// SIMATIC STEP 7 (V5.x) project PLC_PKS
// CPU: CPU 315-2 PN/DP
// station: Hardware
// station: SIMATIC 300
// station: P_ADR_BUS
// program: S7 Program(1)

SYMBOL_TABLE
"CV1_pid"	DB 2	FB 2
"COM"	DB 88	DB 88
"COMM"	DB 100	DB 100
"CV1_ctrl"	DB 201	FB 2
"CV6_ctrl"	DB 206	FB 2
"CV7_ctrl"	DB 207	FB 2
"CV8_ctrl"	DB 208	FB 2
"CV9_ctrl"	DB 209	FB 2
"CV10_ctrl"	DB 210	FB 2
"CV11_ctrl"	DB 211	FB 2
"CV12_ctrl"	DB 212	FB 2
"CV13_ctrl"	DB 213	FB 2
"CV14_ctrl"	DB 214	FB 2
"CV15_ctrl"	DB 215	FB 2
"CV16_ctrl"	DB 216	FB 2
"CV17_ctrl"	DB 217	FB 2
"CV18_1_ctrl"	DB 218	FB 2
"CV18_2_ctrl"	DB 219	FB 2
"CV21_ctrl"	DB 221	FB 2
"CV22_ctrl"	DB 222	FB 2
"ctrl_CV23"	DB 223	FB 2
"ctrl_CV24"	DB 224	FB 2
"ctrl_CV25"	DB 225	FB 2
"pid_cv1"	DB 501	FB 58
"pid_cv2"	DB 502	FB 58
"pid_cv6"	DB 506	FB 58
"pid_cv7"	DB 507	FB 58
"pid_cv8"	DB 508	FB 58
"pid_cv9"	DB 509	FB 58
"pid_cv10"	DB 510	FB 58
"pid_cv11"	DB 511	FB 58
"pid_cv12"	DB 512	FB 58
"pid_cv13"	DB 513	FB 58
"pid_cv14"	DB 514	FB 58
"pid_cv15"	DB 515	FB 58
"pid_cv16"	DB 516	FB 58
"pid_cv17"	DB 517	FB 58
"pid_cv18_1"	DB 518	FB 58
"pid_cv18_2"	DB 519	FB 58
"pid_cv21"	DB 521	FB 58
"pid_cv22"	DB 522	FB 58
"pid_cv23"	DB 523	FB 58
"pid_cv24"	DB 524	FB 58
"pid_cv25"	DB 525	FB 58
"Pumps"	FB 1	FB 1
"klapan"	FB 2	FB 2
"Dat_CV_val"	FB 3	FB 3
"TCONT_CP"	FB 58	FB 58	// temperature PID controller with pulse generator and self-tuning
"Dat_Filt"	FC 1	FC 1
"SCALE"	FC 105	FC 105	// Scaling Values
"UNSCALE"	FC 106	FC 106	// Unscaling Values
"MM1_KM"	M 10.0	BOOL
"M1_Man"	M 1424.0	BOOL
"CV1_val"	MW 500	INT
"CV6_val"	MW 502	INT
"CYC_INT5"	OB 35	OB 35	// Cyclic Interrupt 5
"PT201"	PIW 272	INT
"PT203"	PIW 274	INT
"PT202"	PIW 276	INT
"AI4"	PIW 278	INT
"PT205"	PIW 280	INT
"PT207"	PIW 282	INT
"PT206"	PIW 284	INT
"PT208"	PIW 286	INT
"PT209"	PIW 288	INT
"PT211"	PIW 290	INT
"PT210"	PIW 292	INT
"PT212"	PIW 294	INT
"PT213"	PIW 296	INT
"PT215"	PIW 298	INT
"PT214"	PIW 300	INT
"dPT216"	PIW 302	INT
"dPT217"	PIW 312	INT
"dT219"	PIW 314	INT
"dT218"	PIW 316	INT
"LT301"	PIW 318	INT
"LT302"	PIW 320	INT
"LT304"	PIW 322	INT
"LT303"	PIW 324	INT
"PT220"	PIW 326	INT
"LT305"	PIW 328	INT
"CV1"	PQW 276	INT
"CV7"	PQW 282	INT
"CV6"	PQW 284	INT
"CV8"	PQW 286	INT
"CV9"	PQW 288	INT
"CV11"	PQW 290	INT
"CV10"	PQW 292	INT
"CV12"	PQW 294	INT
"CV13"	PQW 296	INT
"CV15"	PQW 298	INT
"CV14"	PQW 300	INT
"CV16"	PQW 302	INT
"CV17"	PQW 304	INT
"CV18_2"	PQW 306	INT
"CV18_1"	PQW 308	INT
"CV19_1"	PQW 310	INT
"CV19_2"	PQW 312	INT
"CV21"	PQW 314	INT
"CV20"	PQW 316	INT
"CV22"	PQW 318	INT
"CV23"	PQW 320	INT
"CV25"	PQW 322	INT
"CV24"	PQW 324	INT
"M1_KM"	Q 0.0	BOOL
"VAT_CV1"	VAT 1	
"VAT_CV17"	VAT 2	
END_SYMBOL_TABLE

FUNCTION_BLOCK "Pumps"	// FB 1
TITLE = управление насосами
//управление насосами М1-КМ, М2-КМ
VERSION : 0.1
VAR
  Bipolar : BOOL ;
  rst_T1 : BOOL ;
  int_C1 : INT ;
  Hi_lim_re : REAL ;
  Low_lim_re : REAL ;
  DAT_re : REAL ;
  DAT_avg : REAL ;
  Dat_f : REAL ;
  dat_re0 : REAL ;
  dat_re1 : REAL ;
  dat_re2 : REAL ;
  dat_re3 : REAL ;
  dat_re4 : REAL ;
  dat_re5 : REAL ;
  dat_re6 : REAL ;
  dat_re7 : REAL ;
  dat_re8 : REAL ;
  dat_re9 : REAL ;
  sum : REAL ;
  DAT_Hi_Lim : DINT ;
  DAT_Low_Lim : DINT ;
  DAT_PIW : INT ;
  Dat_err_lvl : INT ;
  Dat_err : BOOL ;
  Sample : S5TIME ;
  Dat_md : DINT ;
  HI_LVL : REAL ;
  LOW_LVL : REAL ;
END_VAR
VAR_TEMP
  SCL_err : WORD ;
  UNSCL_err : WORD ;
END_VAR
BEGIN
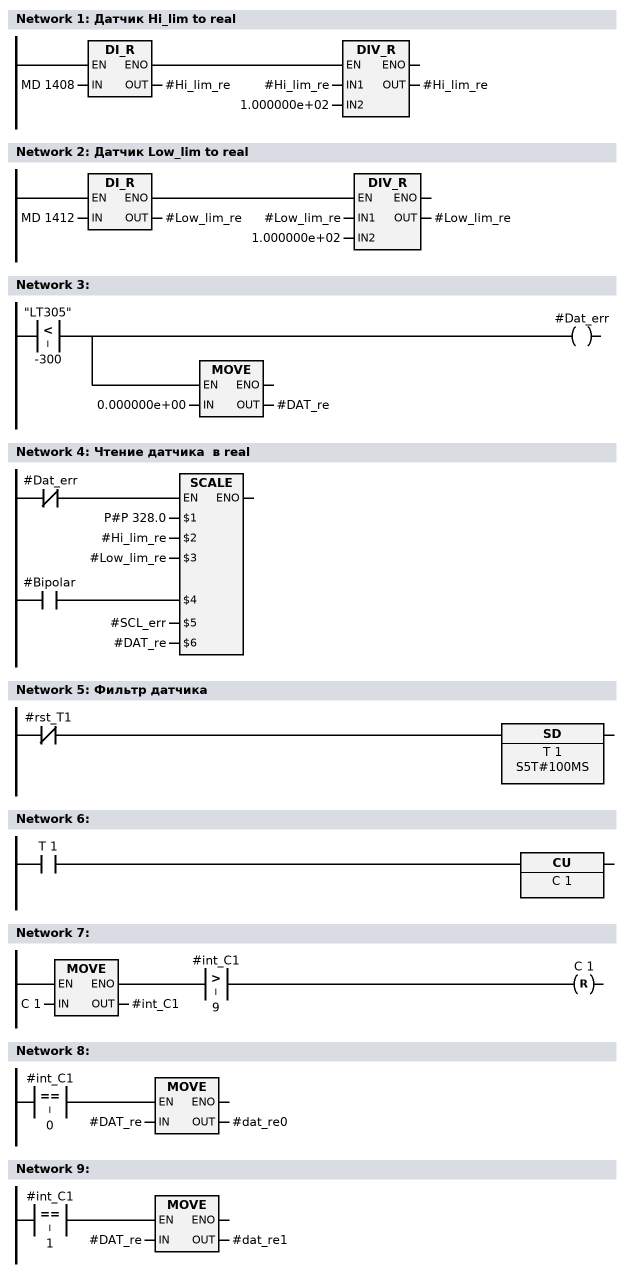
NETWORK
TITLE = Датчик Hi_lim to real
      A(;
      L     MD 1408;
      DTR;
      T     #Hi_lim_re;
      SET;
      SAVE;
      CLR;
      A     BR;
      );
      JNB   _001;
      L     #Hi_lim_re;
      L     1.000000e+02;
      /R;
      T     #Hi_lim_re;
_001: NOP   0;
NETWORK
TITLE = Датчик Low_lim to real
      A(;
      L     MD 1412;
      DTR;
      T     #Low_lim_re;
      SET;
      SAVE;
      CLR;
      A     BR;
      );
      JNB   _002;
      L     #Low_lim_re;
      L     1.000000e+02;
      /R;
      T     #Low_lim_re;
_002: NOP   0;
NETWORK
TITLE =
//Ошибка чтения датчика
      L     "LT305";
      L     -300;
      <I;
      =     L 4.0;
      A     L 4.0;
      BLD   102;
      =     #Dat_err;
      A     L 4.0;
      JNB   _003;
      L     0.000000e+00;
      T     #DAT_re;
_003: NOP   0;
NETWORK
TITLE = Чтение датчика  в real
      A     #Bipolar;
      =     L 4.0;
      BLD   103;
      AN    #Dat_err;
      JNB   _004;
      CALL  "SCALE" (
           $1                       := P#P 328.0,
           $2                       := #Hi_lim_re,
           $3                       := #Low_lim_re,
           $4                       := L 4.0,
           $5                       := #SCL_err,
           $6                       := #DAT_re);
_004: NOP   0;
NETWORK
TITLE = Фильтр датчика
//***************************************************
      AN    #rst_T1;
      L     S5T#100MS;
      SD    T 1;
NETWORK
TITLE =
      A     T 1;
      CU    C 1;
NETWORK
TITLE =
      A(;
      L     C 1;
      T     #int_C1;
      SET;
      SAVE;
      CLR;
      A     BR;
      );
      A(;
      L     #int_C1;
      L     9;
      >I;
      );
      R     C 1;
NETWORK
TITLE =
      A(;
      L     #int_C1;
      L     0;
      ==I;
      );
      JNB   _005;
      L     #DAT_re;
      T     #dat_re0;
_005: NOP   0;
NETWORK
TITLE =
      A(;
      L     #int_C1;
      L     1;
      ==I;
      );
      JNB   _006;
      L     #DAT_re;
      T     #dat_re1;
_006: NOP   0;
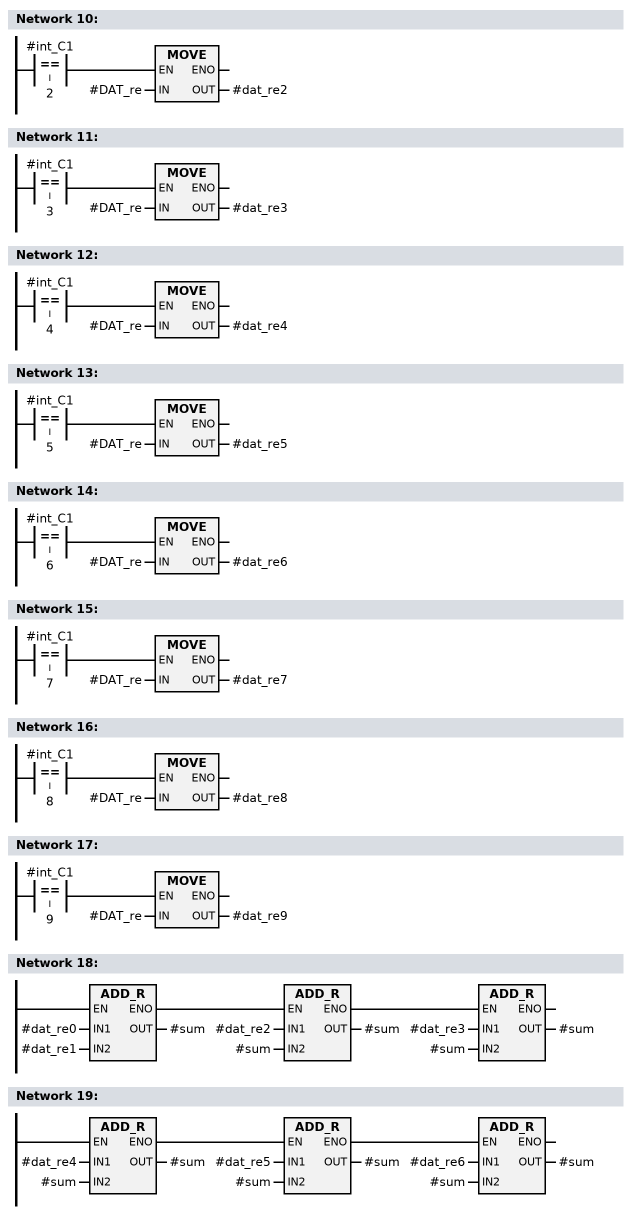
NETWORK
TITLE =
      A(;
      L     #int_C1;
      L     2;
      ==I;
      );
      JNB   _007;
      L     #DAT_re;
      T     #dat_re2;
_007: NOP   0;
NETWORK
TITLE =
      A(;
      L     #int_C1;
      L     3;
      ==I;
      );
      JNB   _008;
      L     #DAT_re;
      T     #dat_re3;
_008: NOP   0;
NETWORK
TITLE =
      A(;
      L     #int_C1;
      L     4;
      ==I;
      );
      JNB   _009;
      L     #DAT_re;
      T     #dat_re4;
_009: NOP   0;
NETWORK
TITLE =
      A(;
      L     #int_C1;
      L     5;
      ==I;
      );
      JNB   _00a;
      L     #DAT_re;
      T     #dat_re5;
_00a: NOP   0;
NETWORK
TITLE =
      A(;
      L     #int_C1;
      L     6;
      ==I;
      );
      JNB   _00b;
      L     #DAT_re;
      T     #dat_re6;
_00b: NOP   0;
NETWORK
TITLE =
      A(;
      L     #int_C1;
      L     7;
      ==I;
      );
      JNB   _00c;
      L     #DAT_re;
      T     #dat_re7;
_00c: NOP   0;
NETWORK
TITLE =
      A(;
      L     #int_C1;
      L     8;
      ==I;
      );
      JNB   _00d;
      L     #DAT_re;
      T     #dat_re8;
_00d: NOP   0;
NETWORK
TITLE =
      A(;
      L     #int_C1;
      L     9;
      ==I;
      );
      JNB   _00e;
      L     #DAT_re;
      T     #dat_re9;
_00e: NOP   0;
NETWORK
TITLE =
      A(;
      A(;
      L     #dat_re0;
      L     #dat_re1;
      +R;
      T     #sum;
      AN    OV;
      SAVE;
      CLR;
      A     BR;
      );
      JNB   _00f;
      L     #dat_re2;
      L     #sum;
      +R;
      T     #sum;
      AN    OV;
      SAVE;
      CLR;
_00f: A     BR;
      );
      JNB   _010;
      L     #dat_re3;
      L     #sum;
      +R;
      T     #sum;
_010: NOP   0;
NETWORK
TITLE =
      A(;
      A(;
      L     #dat_re4;
      L     #sum;
      +R;
      T     #sum;
      AN    OV;
      SAVE;
      CLR;
      A     BR;
      );
      JNB   _011;
      L     #dat_re5;
      L     #sum;
      +R;
      T     #sum;
      AN    OV;
      SAVE;
      CLR;
_011: A     BR;
      );
      JNB   _012;
      L     #dat_re6;
      L     #sum;
      +R;
      T     #sum;
_012: NOP   0;
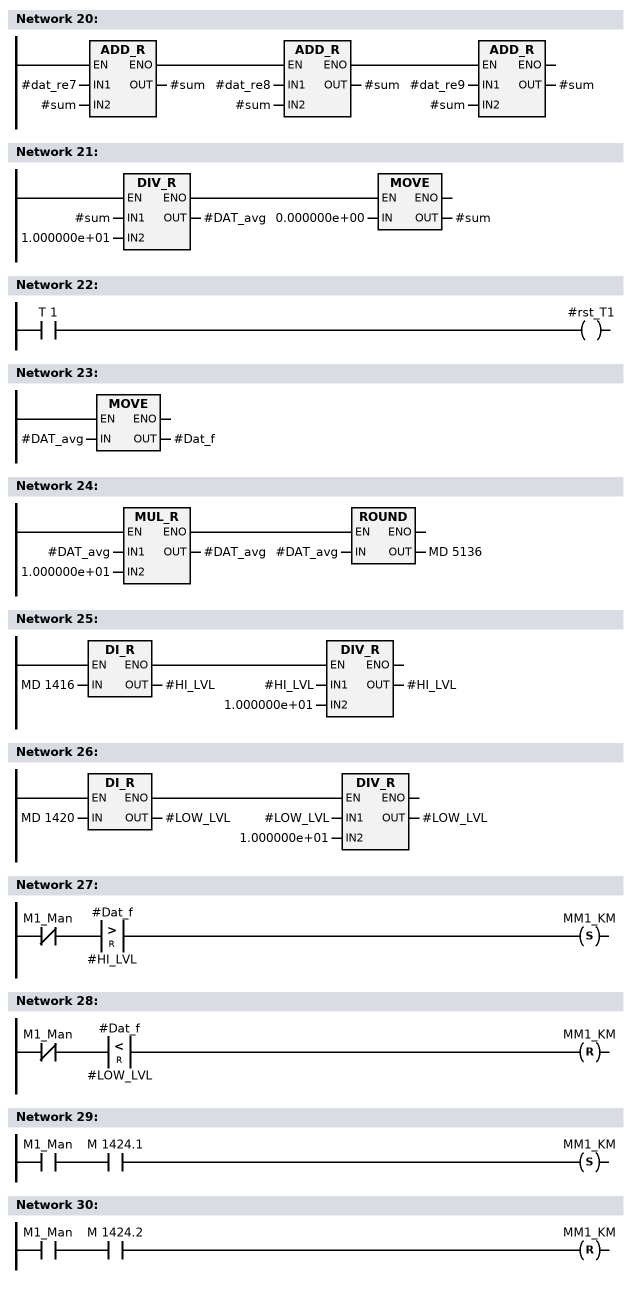
NETWORK
TITLE =
      A(;
      A(;
      L     #dat_re7;
      L     #sum;
      +R;
      T     #sum;
      AN    OV;
      SAVE;
      CLR;
      A     BR;
      );
      JNB   _013;
      L     #dat_re8;
      L     #sum;
      +R;
      T     #sum;
      AN    OV;
      SAVE;
      CLR;
_013: A     BR;
      );
      JNB   _014;
      L     #dat_re9;
      L     #sum;
      +R;
      T     #sum;
_014: NOP   0;
NETWORK
TITLE =
      A(;
      L     #sum;
      L     1.000000e+01;
      /R;
      T     #DAT_avg;
      AN    OV;
      SAVE;
      CLR;
      A     BR;
      );
      JNB   _015;
      L     0.000000e+00;
      T     #sum;
_015: NOP   0;
NETWORK
TITLE =
      A     T 1;
      =     #rst_T1;
NETWORK
TITLE =
      L     #DAT_avg;
      T     #Dat_f;
      NOP   0;
NETWORK
TITLE =
      A(;
      L     #DAT_avg;
      L     1.000000e+01;
      *R;
      T     #DAT_avg;
      AN    OV;
      SAVE;
      CLR;
      A     BR;
      );
      JNB   _016;
      L     #DAT_avg;
      RND;
      T     MD 5136;
_016: NOP   0;
NETWORK
TITLE =
//********************************************************************************
//управление насосом. Верхний уровень в real
      A(;
      L     MD 1416;
      DTR;
      T     #HI_LVL;
      SET;
      SAVE;
      CLR;
      A     BR;
      );
      JNB   _017;
      L     #HI_LVL;
      L     1.000000e+01;
      /R;
      T     #HI_LVL;
_017: NOP   0;
NETWORK
TITLE =
//********************************************************************************
//управление насосом. Нижний уровень в real
      A(;
      L     MD 1420;
      DTR;
      T     #LOW_LVL;
      SET;
      SAVE;
      CLR;
      A     BR;
      );
      JNB   _018;
      L     #LOW_LVL;
      L     1.000000e+01;
      /R;
      T     #LOW_LVL;
_018: NOP   0;
NETWORK
TITLE =
      AN    "M1_Man";
      A(;
      L     #Dat_f;
      L     #HI_LVL;
      >R;
      );
      S     "MM1_KM";
NETWORK
TITLE =
      AN    "M1_Man";
      A(;
      L     #Dat_f;
      L     #LOW_LVL;
      <R;
      );
      R     "MM1_KM";
NETWORK
TITLE =
      A     "M1_Man";
      A     M 1424.1;
      S     "MM1_KM";
NETWORK
TITLE =
      A     "M1_Man";
      A     M 1424.2;
      R     "MM1_KM";
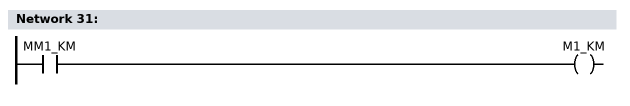
NETWORK
TITLE =
      A     "MM1_KM";
      =     "M1_KM";
END_FUNCTION_BLOCK

FUNCTION_BLOCK "klapan"	// FB 2
TITLE = PID управление клапанами
//PID управление клапанами
VERSION : 0.1
VAR_INPUT
  DAT_PIW : INT ;
  DAT_Hi_Lim : DWORD ;
  DAT_Low_Lim : DWORD ;
  Dat_err_lvl : INT ;
  P_dw : DWORD ;
  I_dw : DWORD ;
  D_dw : DWORD ;
  TASK_dw : DWORD ;
  PID_LMN : REAL ;
  Pulse_Sample : BOOL ;
END_VAR
VAR_OUTPUT
  Dat_err : BOOL ;
  DAT_f : REAL ;
  TASK_pid : REAL ;
  P_pid : REAL ;
  I_pid : REAL ;
  D_pid : REAL ;
  CV_PQW : INT ;
  DAT_md : DWORD ;
  CV_md : DWORD ;
END_VAR
VAR
  Bipolar : BOOL ;
  rst_T0 : BOOL ;
  int_C0 : INT ;
  Hi_lim_re : REAL ;
  Low_lim_re : REAL ;
  DAT_re : REAL ;
  DAT_avg : REAL ;
  dat_re0 : REAL ;
  dat_re1 : REAL ;
  dat_re2 : REAL ;
  dat_re3 : REAL ;
  dat_re4 : REAL ;
  dat_re5 : REAL ;
  dat_re6 : REAL ;
  dat_re7 : REAL ;
  dat_re8 : REAL ;
  dat_re9 : REAL ;
  sum : REAL ;
  CV_val : INT ;
  Count_Sample : INT ;
  OldPulseSample : BOOL ;
  Pulse_Scan : BOOL ;
END_VAR
VAR_TEMP
  SCL_err : WORD ;
  UNSCL_err : WORD ;
END_VAR
BEGIN
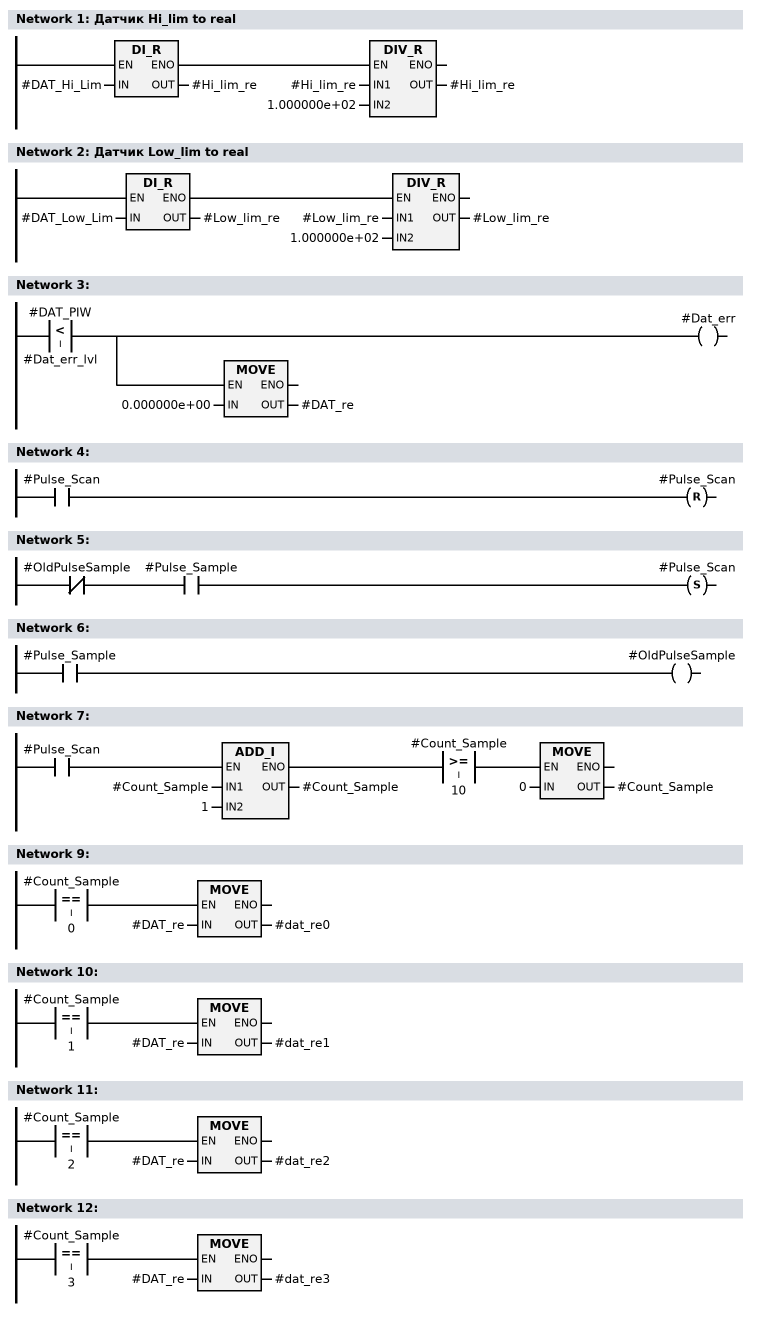
NETWORK
TITLE = Датчик Hi_lim to real
      A(;
      L     #DAT_Hi_Lim;
      DTR;
      T     #Hi_lim_re;
      SET;
      SAVE;
      CLR;
      A     BR;
      );
      JNB   _001;
      L     #Hi_lim_re;
      L     1.000000e+02;
      /R;
      T     #Hi_lim_re;
_001: NOP   0;
NETWORK
TITLE = Датчик Low_lim to real
      A(;
      L     #DAT_Low_Lim;
      DTR;
      T     #Low_lim_re;
      SET;
      SAVE;
      CLR;
      A     BR;
      );
      JNB   _002;
      L     #Low_lim_re;
      L     1.000000e+02;
      /R;
      T     #Low_lim_re;
_002: NOP   0;
NETWORK
TITLE =
//Ошибка чтения датчика
      L     #DAT_PIW;
      L     #Dat_err_lvl;
      <I;
      =     L 4.0;
      A     L 4.0;
      BLD   102;
      =     #Dat_err;
      A     L 4.0;
      JNB   _003;
      L     0.000000e+00;
      T     #DAT_re;
_003: NOP   0;
NETWORK
TITLE =
      A     #Pulse_Scan;
      R     #Pulse_Scan;
NETWORK
TITLE =
      AN    #OldPulseSample;
      A     #Pulse_Sample;
      S     #Pulse_Scan;
NETWORK
TITLE =
      A     #Pulse_Sample;
      =     #OldPulseSample;
NETWORK
TITLE =
      A(;
      A     #Pulse_Scan;
      JNB   _004;
      L     #Count_Sample;
      L     1;
      +I;
      T     #Count_Sample;
      AN    OV;
      SAVE;
      CLR;
_004: A     BR;
      );
      A(;
      L     #Count_Sample;
      L     10;
      >=I;
      );
      JNB   _005;
      L     0;
      T     #Count_Sample;
_005: NOP   0;
NETWORK
TITLE = Чтение датчика (MPa)x10 = Bar
      A(;
      A     #Bipolar;
      =     L 4.0;
      BLD   103;
      AN    #Dat_err;
      JNB   _006;
      CALL  "SCALE" (
           $1                       := #DAT_PIW,
           $2                       := #Hi_lim_re,
           $3                       := #Low_lim_re,
           $4                       := L 4.0,
           $5                       := #SCL_err,
           $6                       := #DAT_re);
_006: A     BR;
      );
      JNB   _007;
      L     #DAT_re;
      L     1.000000e+01;
      *R;
      T     #DAT_re;
_007: NOP   0;
NETWORK
TITLE =
      A(;
      L     #Count_Sample;
      L     0;
      ==I;
      );
      JNB   _008;
      L     #DAT_re;
      T     #dat_re0;
_008: NOP   0;
NETWORK
TITLE =
      A(;
      L     #Count_Sample;
      L     1;
      ==I;
      );
      JNB   _009;
      L     #DAT_re;
      T     #dat_re1;
_009: NOP   0;
NETWORK
TITLE =
      A(;
      L     #Count_Sample;
      L     2;
      ==I;
      );
      JNB   _00a;
      L     #DAT_re;
      T     #dat_re2;
_00a: NOP   0;
NETWORK
TITLE =
      A(;
      L     #Count_Sample;
      L     3;
      ==I;
      );
      JNB   _00b;
      L     #DAT_re;
      T     #dat_re3;
_00b: NOP   0;
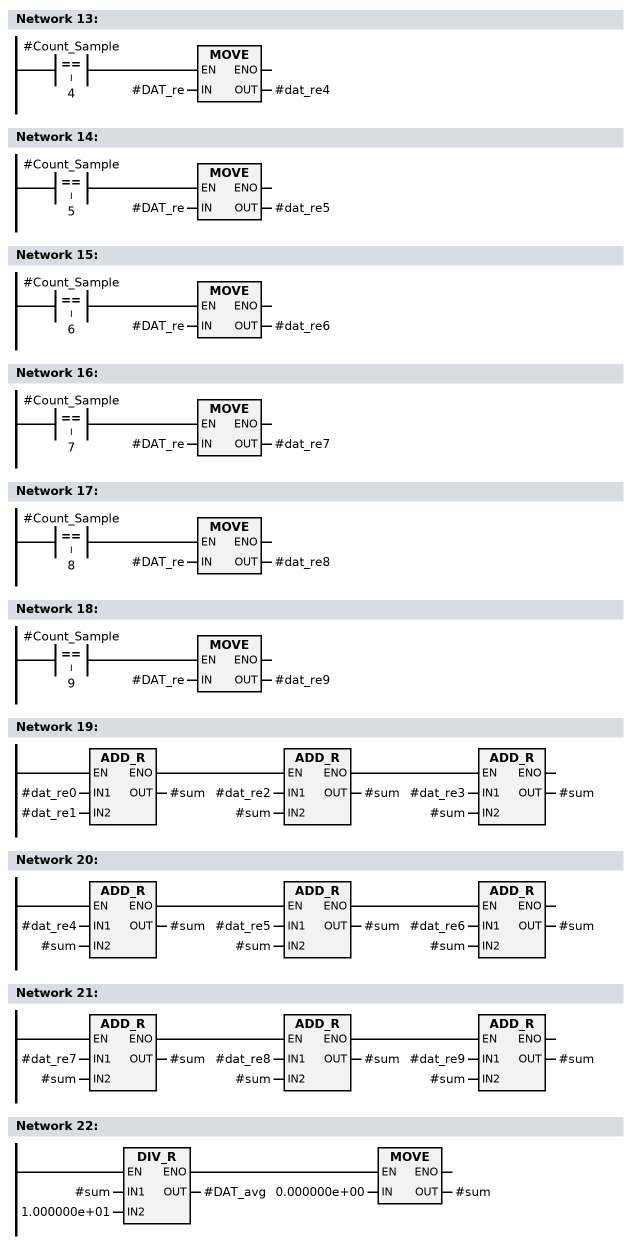
NETWORK
TITLE =
      A(;
      L     #Count_Sample;
      L     4;
      ==I;
      );
      JNB   _00c;
      L     #DAT_re;
      T     #dat_re4;
_00c: NOP   0;
NETWORK
TITLE =
      A(;
      L     #Count_Sample;
      L     5;
      ==I;
      );
      JNB   _00d;
      L     #DAT_re;
      T     #dat_re5;
_00d: NOP   0;
NETWORK
TITLE =
      A(;
      L     #Count_Sample;
      L     6;
      ==I;
      );
      JNB   _00e;
      L     #DAT_re;
      T     #dat_re6;
_00e: NOP   0;
NETWORK
TITLE =
      A(;
      L     #Count_Sample;
      L     7;
      ==I;
      );
      JNB   _00f;
      L     #DAT_re;
      T     #dat_re7;
_00f: NOP   0;
NETWORK
TITLE =
      A(;
      L     #Count_Sample;
      L     8;
      ==I;
      );
      JNB   _010;
      L     #DAT_re;
      T     #dat_re8;
_010: NOP   0;
NETWORK
TITLE =
      A(;
      L     #Count_Sample;
      L     9;
      ==I;
      );
      JNB   _011;
      L     #DAT_re;
      T     #dat_re9;
_011: NOP   0;
NETWORK
TITLE =
      A(;
      A(;
      L     #dat_re0;
      L     #dat_re1;
      +R;
      T     #sum;
      AN    OV;
      SAVE;
      CLR;
      A     BR;
      );
      JNB   _012;
      L     #dat_re2;
      L     #sum;
      +R;
      T     #sum;
      AN    OV;
      SAVE;
      CLR;
_012: A     BR;
      );
      JNB   _013;
      L     #dat_re3;
      L     #sum;
      +R;
      T     #sum;
_013: NOP   0;
NETWORK
TITLE =
      A(;
      A(;
      L     #dat_re4;
      L     #sum;
      +R;
      T     #sum;
      AN    OV;
      SAVE;
      CLR;
      A     BR;
      );
      JNB   _014;
      L     #dat_re5;
      L     #sum;
      +R;
      T     #sum;
      AN    OV;
      SAVE;
      CLR;
_014: A     BR;
      );
      JNB   _015;
      L     #dat_re6;
      L     #sum;
      +R;
      T     #sum;
_015: NOP   0;
NETWORK
TITLE =
      A(;
      A(;
      L     #dat_re7;
      L     #sum;
      +R;
      T     #sum;
      AN    OV;
      SAVE;
      CLR;
      A     BR;
      );
      JNB   _016;
      L     #dat_re8;
      L     #sum;
      +R;
      T     #sum;
      AN    OV;
      SAVE;
      CLR;
_016: A     BR;
      );
      JNB   _01d;
      L     #dat_re9;
      L     #sum;
      +R;
      T     #sum;
_01d: NOP   0;
NETWORK
TITLE =
      A(;
      L     #sum;
      L     1.000000e+01;
      /R;
      T     #DAT_avg;
      AN    OV;
      SAVE;
      CLR;
      A     BR;
      );
      JNB   _01f;
      L     0.000000e+00;
      T     #sum;
_01f: NOP   0;
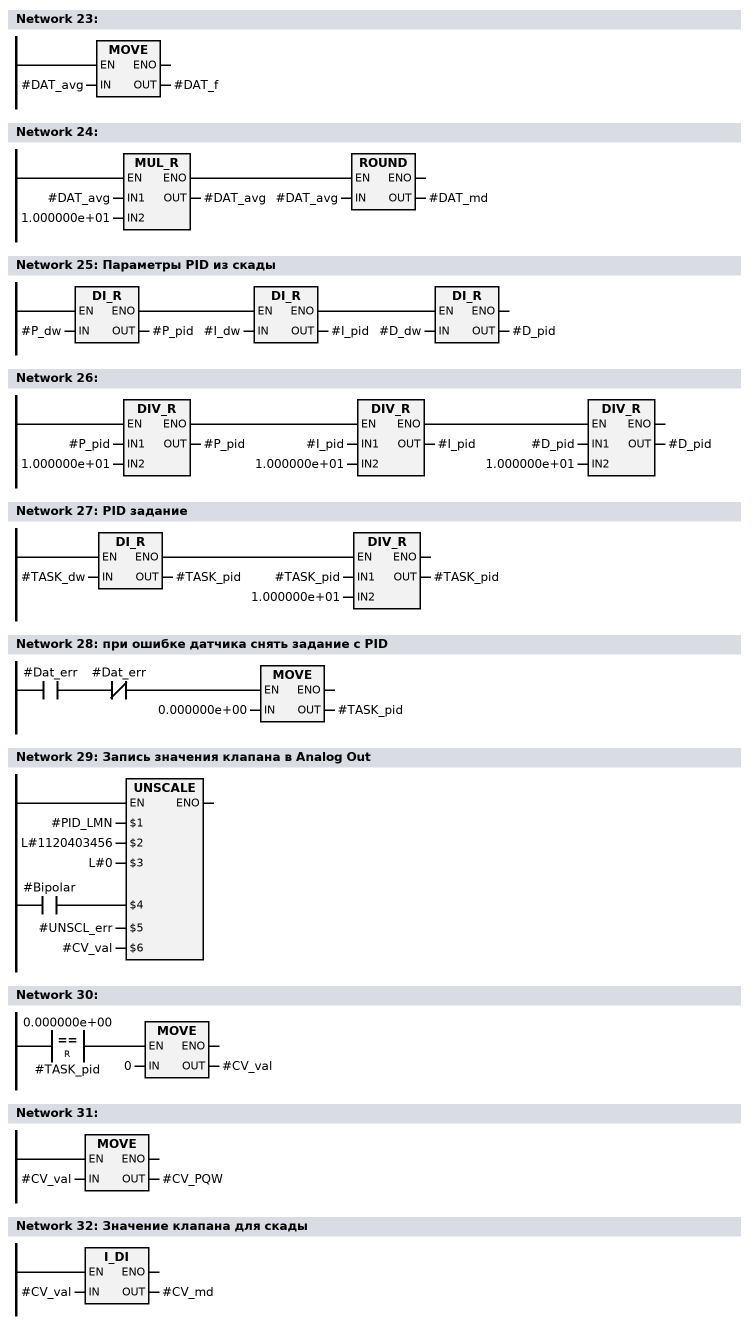
NETWORK
TITLE =
      L     #DAT_avg;
      T     #DAT_f;
      NOP   0;
NETWORK
TITLE =
      A(;
      L     #DAT_avg;
      L     1.000000e+01;
      *R;
      T     #DAT_avg;
      AN    OV;
      SAVE;
      CLR;
      A     BR;
      );
      JNB   _017;
      L     #DAT_avg;
      RND;
      T     #DAT_md;
_017: NOP   0;
NETWORK
TITLE = Параметры PID из скады
//********************************************************************************
//
      A(;
      A(;
      L     #P_dw;
      DTR;
      T     #P_pid;
      SET;
      SAVE;
      CLR;
      A     BR;
      );
      JNB   _018;
      L     #I_dw;
      DTR;
      T     #I_pid;
      SET;
      SAVE;
      CLR;
_018: A     BR;
      );
      JNB   _019;
      L     #D_dw;
      DTR;
      T     #D_pid;
_019: NOP   0;
NETWORK
TITLE =
      A(;
      A(;
      L     #P_pid;
      L     1.000000e+01;
      /R;
      T     #P_pid;
      AN    OV;
      SAVE;
      CLR;
      A     BR;
      );
      JNB   _01a;
      L     #I_pid;
      L     1.000000e+01;
      /R;
      T     #I_pid;
      AN    OV;
      SAVE;
      CLR;
_01a: A     BR;
      );
      JNB   _01b;
      L     #D_pid;
      L     1.000000e+01;
      /R;
      T     #D_pid;
_01b: NOP   0;
NETWORK
TITLE = PID задание
      A(;
      L     #TASK_dw;
      DTR;
      T     #TASK_pid;
      SET;
      SAVE;
      CLR;
      A     BR;
      );
      JNB   _01c;
      L     #TASK_pid;
      L     1.000000e+01;
      /R;
      T     #TASK_pid;
_01c: NOP   0;
NETWORK
TITLE = при ошибке датчика снять задание с PID
      A     #Dat_err;
      AN    #Dat_err;
      JNB   _020;
      L     0.000000e+00;
      T     #TASK_pid;
_020: NOP   0;
NETWORK
TITLE = Запись значения клапана в Analog Out
      A     #Bipolar;
      =     L 4.0;
      BLD   103;
      CALL  "UNSCALE" (
           $1                       := #PID_LMN,
           $2                       := L#1120403456,
           $3                       := L#0,
           $4                       := L 4.0,
           $5                       := #UNSCL_err,
           $6                       := #CV_val);
      NOP   0;
NETWORK
TITLE =
//Если задание 0, то записать 0 в значение клапана
      A(;
      L     0.000000e+00;
      L     #TASK_pid;
      ==R;
      );
      JNB   _01e;
      L     0;
      T     #CV_val;
_01e: NOP   0;
NETWORK
TITLE =
      L     #CV_val;
      T     #CV_PQW;
      NOP   0;
NETWORK
TITLE = Значение клапана для скады
      L     #CV_val;
      ITD;
      T     #CV_md;
      NOP   0;
END_FUNCTION_BLOCK

FUNCTION_BLOCK "Dat_CV_val"	// FB 3
//значення датчиків і клапанів для SCADA та HMI
VERSION : 0.1
VAR
  cv_re : REAL ;
END_VAR
BEGIN
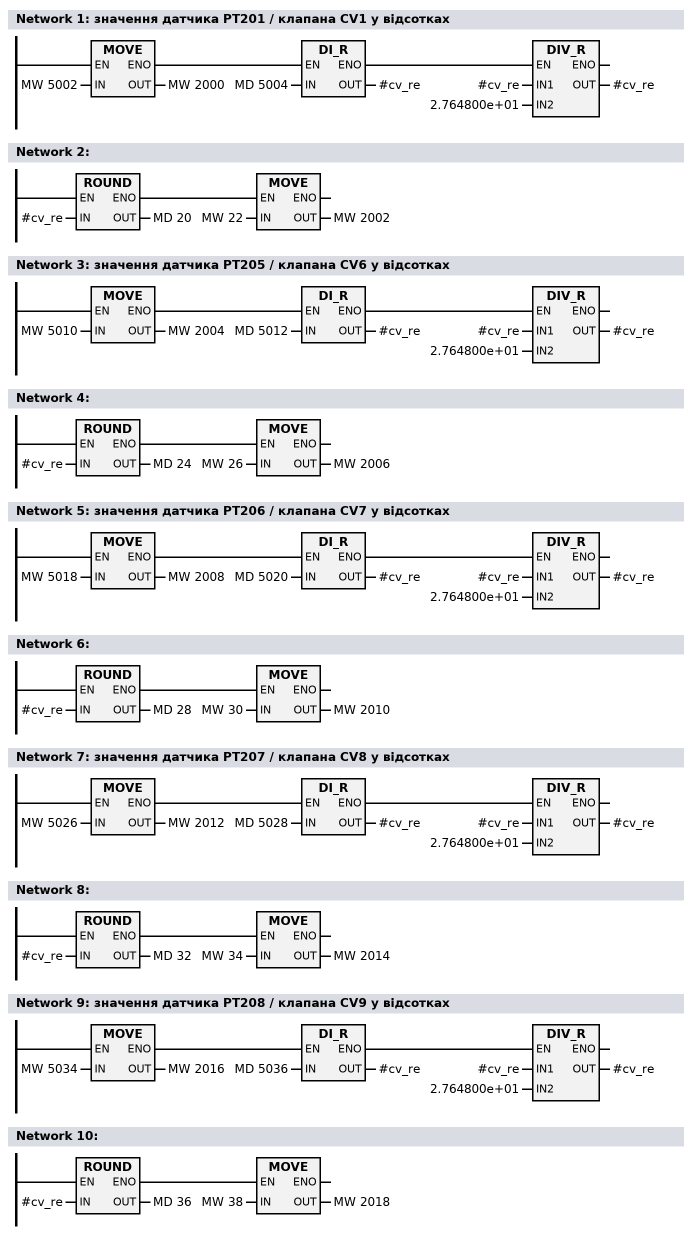
NETWORK
TITLE = значення датчика PT201 / клапана CV1 у відсотках
      A(;
      A(;
      L     MW 5002;
      T     MW 2000;
      SET;
      SAVE;
      CLR;
      A     BR;
      );
      JNB   _001;
      L     MD 5004;
      DTR;
      T     #cv_re;
      SET;
      SAVE;
      CLR;
_001: A     BR;
      );
      JNB   _002;
      L     #cv_re;
      L     2.764800e+01;
      /R;
      T     #cv_re;
_002: NOP   0;
NETWORK
TITLE =
      A(;
      L     #cv_re;
      RND;
      T     MD 20;
      AN    OV;
      SAVE;
      CLR;
      A     BR;
      );
      JNB   _003;
      L     MW 22;
      T     MW 2002;
_003: NOP   0;
NETWORK
TITLE = значення датчика PT205 / клапана CV6 у відсотках
      A(;
      A(;
      L     MW 5010;
      T     MW 2004;
      SET;
      SAVE;
      CLR;
      A     BR;
      );
      JNB   _004;
      L     MD 5012;
      DTR;
      T     #cv_re;
      SET;
      SAVE;
      CLR;
_004: A     BR;
      );
      JNB   _005;
      L     #cv_re;
      L     2.764800e+01;
      /R;
      T     #cv_re;
_005: NOP   0;
NETWORK
TITLE =
      A(;
      L     #cv_re;
      RND;
      T     MD 24;
      AN    OV;
      SAVE;
      CLR;
      A     BR;
      );
      JNB   _006;
      L     MW 26;
      T     MW 2006;
_006: NOP   0;
NETWORK
TITLE = значення датчика PT206 / клапана CV7 у відсотках
      A(;
      A(;
      L     MW 5018;
      T     MW 2008;
      SET;
      SAVE;
      CLR;
      A     BR;
      );
      JNB   _007;
      L     MD 5020;
      DTR;
      T     #cv_re;
      SET;
      SAVE;
      CLR;
_007: A     BR;
      );
      JNB   _008;
      L     #cv_re;
      L     2.764800e+01;
      /R;
      T     #cv_re;
_008: NOP   0;
NETWORK
TITLE =
      A(;
      L     #cv_re;
      RND;
      T     MD 28;
      AN    OV;
      SAVE;
      CLR;
      A     BR;
      );
      JNB   _009;
      L     MW 30;
      T     MW 2010;
_009: NOP   0;
NETWORK
TITLE = значення датчика PT207 / клапана CV8 у відсотках
      A(;
      A(;
      L     MW 5026;
      T     MW 2012;
      SET;
      SAVE;
      CLR;
      A     BR;
      );
      JNB   _00a;
      L     MD 5028;
      DTR;
      T     #cv_re;
      SET;
      SAVE;
      CLR;
_00a: A     BR;
      );
      JNB   _00b;
      L     #cv_re;
      L     2.764800e+01;
      /R;
      T     #cv_re;
_00b: NOP   0;
NETWORK
TITLE =
      A(;
      L     #cv_re;
      RND;
      T     MD 32;
      AN    OV;
      SAVE;
      CLR;
      A     BR;
      );
      JNB   _00c;
      L     MW 34;
      T     MW 2014;
_00c: NOP   0;
NETWORK
TITLE = значення датчика PT208 / клапана CV9 у відсотках
      A(;
      A(;
      L     MW 5034;
      T     MW 2016;
      SET;
      SAVE;
      CLR;
      A     BR;
      );
      JNB   _00d;
      L     MD 5036;
      DTR;
      T     #cv_re;
      SET;
      SAVE;
      CLR;
_00d: A     BR;
      );
      JNB   _00e;
      L     #cv_re;
      L     2.764800e+01;
      /R;
      T     #cv_re;
_00e: NOP   0;
NETWORK
TITLE =
      A(;
      L     #cv_re;
      RND;
      T     MD 36;
      AN    OV;
      SAVE;
      CLR;
      A     BR;
      );
      JNB   _00f;
      L     MW 38;
      T     MW 2018;
_00f: NOP   0;
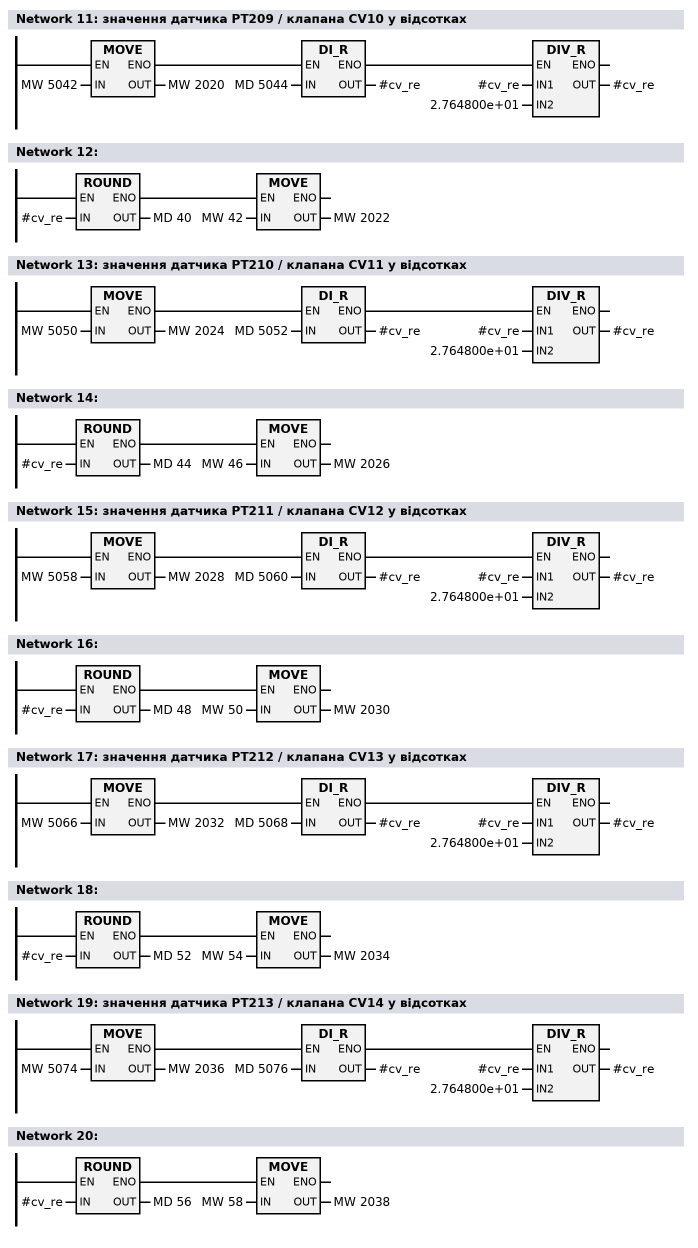
NETWORK
TITLE = значення датчика PT209 / клапана CV10 у відсотках
      A(;
      A(;
      L     MW 5042;
      T     MW 2020;
      SET;
      SAVE;
      CLR;
      A     BR;
      );
      JNB   _010;
      L     MD 5044;
      DTR;
      T     #cv_re;
      SET;
      SAVE;
      CLR;
_010: A     BR;
      );
      JNB   _011;
      L     #cv_re;
      L     2.764800e+01;
      /R;
      T     #cv_re;
_011: NOP   0;
NETWORK
TITLE =
      A(;
      L     #cv_re;
      RND;
      T     MD 40;
      AN    OV;
      SAVE;
      CLR;
      A     BR;
      );
      JNB   _012;
      L     MW 42;
      T     MW 2022;
_012: NOP   0;
NETWORK
TITLE = значення датчика PT210 / клапана CV11 у відсотках
      A(;
      A(;
      L     MW 5050;
      T     MW 2024;
      SET;
      SAVE;
      CLR;
      A     BR;
      );
      JNB   _013;
      L     MD 5052;
      DTR;
      T     #cv_re;
      SET;
      SAVE;
      CLR;
_013: A     BR;
      );
      JNB   _014;
      L     #cv_re;
      L     2.764800e+01;
      /R;
      T     #cv_re;
_014: NOP   0;
NETWORK
TITLE =
      A(;
      L     #cv_re;
      RND;
      T     MD 44;
      AN    OV;
      SAVE;
      CLR;
      A     BR;
      );
      JNB   _015;
      L     MW 46;
      T     MW 2026;
_015: NOP   0;
NETWORK
TITLE = значення датчика PT211 / клапана CV12 у відсотках
      A(;
      A(;
      L     MW 5058;
      T     MW 2028;
      SET;
      SAVE;
      CLR;
      A     BR;
      );
      JNB   _016;
      L     MD 5060;
      DTR;
      T     #cv_re;
      SET;
      SAVE;
      CLR;
_016: A     BR;
      );
      JNB   _017;
      L     #cv_re;
      L     2.764800e+01;
      /R;
      T     #cv_re;
_017: NOP   0;
NETWORK
TITLE =
      A(;
      L     #cv_re;
      RND;
      T     MD 48;
      AN    OV;
      SAVE;
      CLR;
      A     BR;
      );
      JNB   _018;
      L     MW 50;
      T     MW 2030;
_018: NOP   0;
NETWORK
TITLE = значення датчика PT212 / клапана CV13 у відсотках
      A(;
      A(;
      L     MW 5066;
      T     MW 2032;
      SET;
      SAVE;
      CLR;
      A     BR;
      );
      JNB   _019;
      L     MD 5068;
      DTR;
      T     #cv_re;
      SET;
      SAVE;
      CLR;
_019: A     BR;
      );
      JNB   _01a;
      L     #cv_re;
      L     2.764800e+01;
      /R;
      T     #cv_re;
_01a: NOP   0;
NETWORK
TITLE =
      A(;
      L     #cv_re;
      RND;
      T     MD 52;
      AN    OV;
      SAVE;
      CLR;
      A     BR;
      );
      JNB   _01b;
      L     MW 54;
      T     MW 2034;
_01b: NOP   0;
NETWORK
TITLE = значення датчика PT213 / клапана CV14 у відсотках
      A(;
      A(;
      L     MW 5074;
      T     MW 2036;
      SET;
      SAVE;
      CLR;
      A     BR;
      );
      JNB   _01c;
      L     MD 5076;
      DTR;
      T     #cv_re;
      SET;
      SAVE;
      CLR;
_01c: A     BR;
      );
      JNB   _01d;
      L     #cv_re;
      L     2.764800e+01;
      /R;
      T     #cv_re;
_01d: NOP   0;
NETWORK
TITLE =
      A(;
      L     #cv_re;
      RND;
      T     MD 56;
      AN    OV;
      SAVE;
      CLR;
      A     BR;
      );
      JNB   _01e;
      L     MW 58;
      T     MW 2038;
_01e: NOP   0;
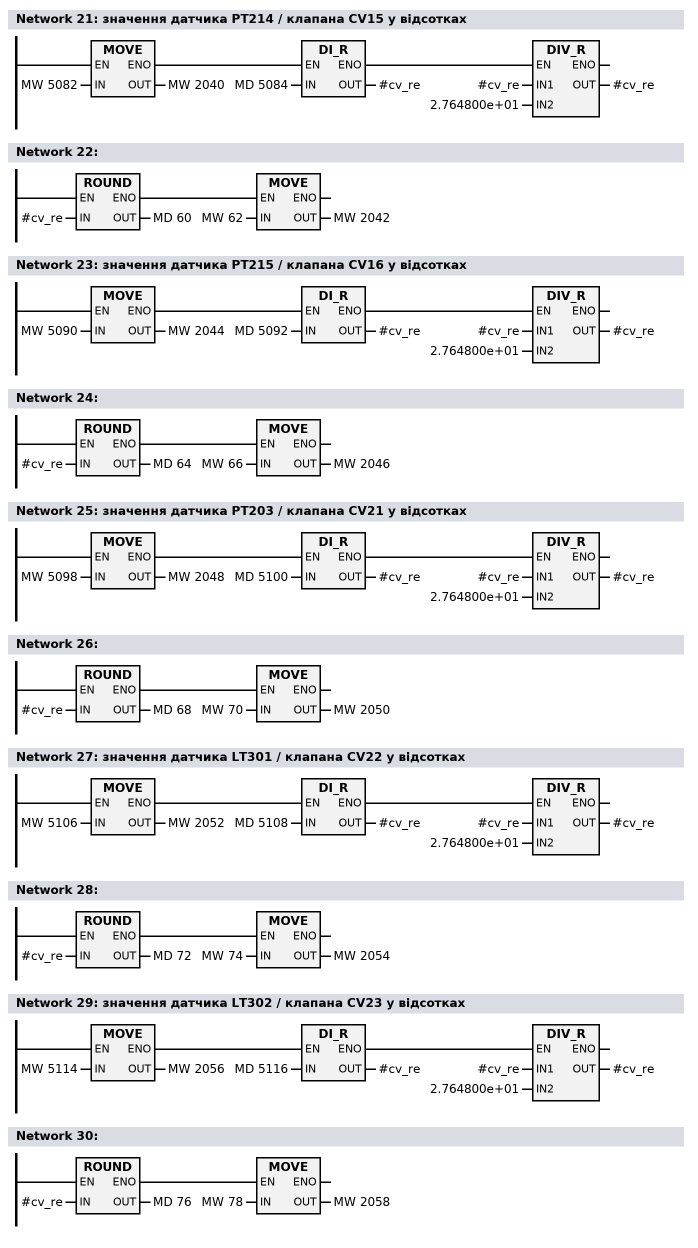
NETWORK
TITLE = значення датчика PT214 / клапана CV15 у відсотках
      A(;
      A(;
      L     MW 5082;
      T     MW 2040;
      SET;
      SAVE;
      CLR;
      A     BR;
      );
      JNB   _01f;
      L     MD 5084;
      DTR;
      T     #cv_re;
      SET;
      SAVE;
      CLR;
_01f: A     BR;
      );
      JNB   _020;
      L     #cv_re;
      L     2.764800e+01;
      /R;
      T     #cv_re;
_020: NOP   0;
NETWORK
TITLE =
      A(;
      L     #cv_re;
      RND;
      T     MD 60;
      AN    OV;
      SAVE;
      CLR;
      A     BR;
      );
      JNB   _021;
      L     MW 62;
      T     MW 2042;
_021: NOP   0;
NETWORK
TITLE = значення датчика PT215 / клапана CV16 у відсотках
      A(;
      A(;
      L     MW 5090;
      T     MW 2044;
      SET;
      SAVE;
      CLR;
      A     BR;
      );
      JNB   _022;
      L     MD 5092;
      DTR;
      T     #cv_re;
      SET;
      SAVE;
      CLR;
_022: A     BR;
      );
      JNB   _023;
      L     #cv_re;
      L     2.764800e+01;
      /R;
      T     #cv_re;
_023: NOP   0;
NETWORK
TITLE =
      A(;
      L     #cv_re;
      RND;
      T     MD 64;
      AN    OV;
      SAVE;
      CLR;
      A     BR;
      );
      JNB   _024;
      L     MW 66;
      T     MW 2046;
_024: NOP   0;
NETWORK
TITLE = значення датчика PT203 / клапана CV21 у відсотках
      A(;
      A(;
      L     MW 5098;
      T     MW 2048;
      SET;
      SAVE;
      CLR;
      A     BR;
      );
      JNB   _025;
      L     MD 5100;
      DTR;
      T     #cv_re;
      SET;
      SAVE;
      CLR;
_025: A     BR;
      );
      JNB   _026;
      L     #cv_re;
      L     2.764800e+01;
      /R;
      T     #cv_re;
_026: NOP   0;
NETWORK
TITLE =
      A(;
      L     #cv_re;
      RND;
      T     MD 68;
      AN    OV;
      SAVE;
      CLR;
      A     BR;
      );
      JNB   _027;
      L     MW 70;
      T     MW 2050;
_027: NOP   0;
NETWORK
TITLE = значення датчика LT301 / клапана CV22 у відсотках
      A(;
      A(;
      L     MW 5106;
      T     MW 2052;
      SET;
      SAVE;
      CLR;
      A     BR;
      );
      JNB   _028;
      L     MD 5108;
      DTR;
      T     #cv_re;
      SET;
      SAVE;
      CLR;
_028: A     BR;
      );
      JNB   _029;
      L     #cv_re;
      L     2.764800e+01;
      /R;
      T     #cv_re;
_029: NOP   0;
NETWORK
TITLE =
      A(;
      L     #cv_re;
      RND;
      T     MD 72;
      AN    OV;
      SAVE;
      CLR;
      A     BR;
      );
      JNB   _02a;
      L     MW 74;
      T     MW 2054;
_02a: NOP   0;
NETWORK
TITLE = значення датчика LT302 / клапана CV23 у відсотках
      A(;
      A(;
      L     MW 5114;
      T     MW 2056;
      SET;
      SAVE;
      CLR;
      A     BR;
      );
      JNB   _02b;
      L     MD 5116;
      DTR;
      T     #cv_re;
      SET;
      SAVE;
      CLR;
_02b: A     BR;
      );
      JNB   _02c;
      L     #cv_re;
      L     2.764800e+01;
      /R;
      T     #cv_re;
_02c: NOP   0;
NETWORK
TITLE =
      A(;
      L     #cv_re;
      RND;
      T     MD 76;
      AN    OV;
      SAVE;
      CLR;
      A     BR;
      );
      JNB   _02d;
      L     MW 78;
      T     MW 2058;
_02d: NOP   0;
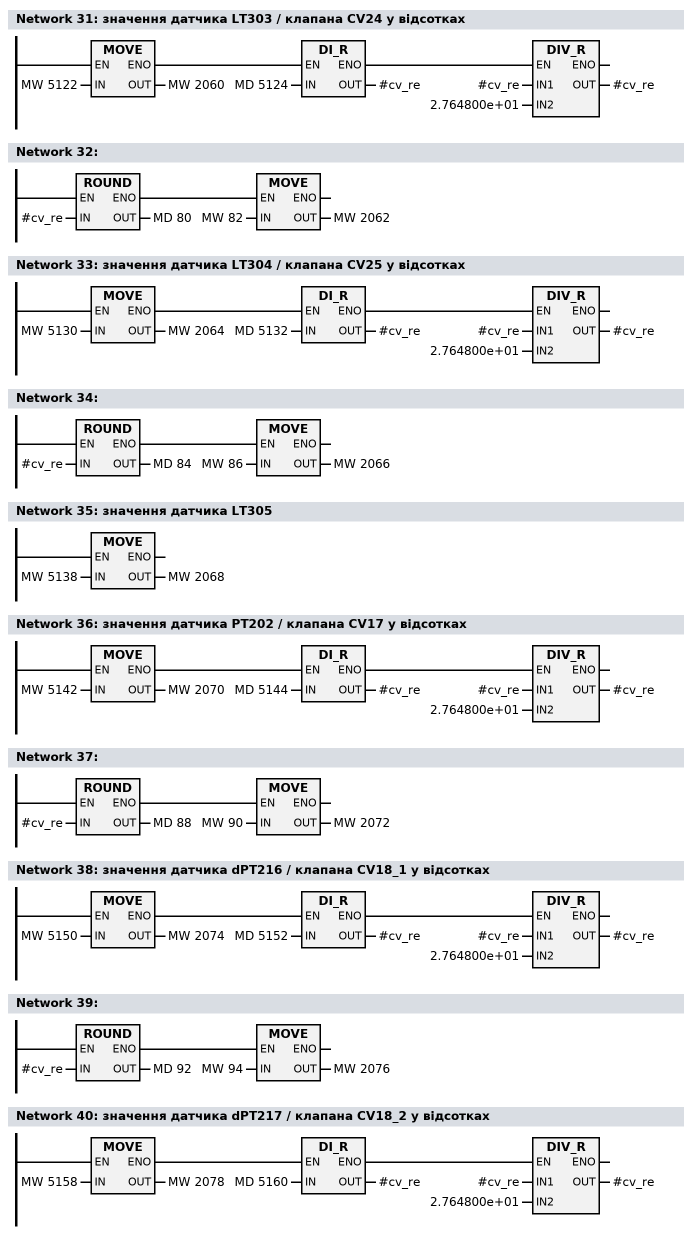
NETWORK
TITLE = значення датчика LT303 / клапана CV24 у відсотках
      A(;
      A(;
      L     MW 5122;
      T     MW 2060;
      SET;
      SAVE;
      CLR;
      A     BR;
      );
      JNB   _02e;
      L     MD 5124;
      DTR;
      T     #cv_re;
      SET;
      SAVE;
      CLR;
_02e: A     BR;
      );
      JNB   _02f;
      L     #cv_re;
      L     2.764800e+01;
      /R;
      T     #cv_re;
_02f: NOP   0;
NETWORK
TITLE =
      A(;
      L     #cv_re;
      RND;
      T     MD 80;
      AN    OV;
      SAVE;
      CLR;
      A     BR;
      );
      JNB   _030;
      L     MW 82;
      T     MW 2062;
_030: NOP   0;
NETWORK
TITLE = значення датчика LT304 / клапана CV25 у відсотках
      A(;
      A(;
      L     MW 5130;
      T     MW 2064;
      SET;
      SAVE;
      CLR;
      A     BR;
      );
      JNB   _031;
      L     MD 5132;
      DTR;
      T     #cv_re;
      SET;
      SAVE;
      CLR;
_031: A     BR;
      );
      JNB   _032;
      L     #cv_re;
      L     2.764800e+01;
      /R;
      T     #cv_re;
_032: NOP   0;
NETWORK
TITLE =
      A(;
      L     #cv_re;
      RND;
      T     MD 84;
      AN    OV;
      SAVE;
      CLR;
      A     BR;
      );
      JNB   _033;
      L     MW 86;
      T     MW 2066;
_033: NOP   0;
NETWORK
TITLE = значення датчика LT305
      L     MW 5138;
      T     MW 2068;
      NOP   0;
NETWORK
TITLE = значення датчика PT202 / клапана CV17 у відсотках
      A(;
      A(;
      L     MW 5142;
      T     MW 2070;
      SET;
      SAVE;
      CLR;
      A     BR;
      );
      JNB   _034;
      L     MD 5144;
      DTR;
      T     #cv_re;
      SET;
      SAVE;
      CLR;
_034: A     BR;
      );
      JNB   _035;
      L     #cv_re;
      L     2.764800e+01;
      /R;
      T     #cv_re;
_035: NOP   0;
NETWORK
TITLE =
      A(;
      L     #cv_re;
      RND;
      T     MD 88;
      AN    OV;
      SAVE;
      CLR;
      A     BR;
      );
      JNB   _036;
      L     MW 90;
      T     MW 2072;
_036: NOP   0;
NETWORK
TITLE = значення датчика dPT216 / клапана CV18_1 у відсотках
      A(;
      A(;
      L     MW 5150;
      T     MW 2074;
      SET;
      SAVE;
      CLR;
      A     BR;
      );
      JNB   _037;
      L     MD 5152;
      DTR;
      T     #cv_re;
      SET;
      SAVE;
      CLR;
_037: A     BR;
      );
      JNB   _038;
      L     #cv_re;
      L     2.764800e+01;
      /R;
      T     #cv_re;
_038: NOP   0;
NETWORK
TITLE =
      A(;
      L     #cv_re;
      RND;
      T     MD 92;
      AN    OV;
      SAVE;
      CLR;
      A     BR;
      );
      JNB   _039;
      L     MW 94;
      T     MW 2076;
_039: NOP   0;
NETWORK
TITLE = значення датчика dPT217 / клапана CV18_2 у відсотках
      A(;
      A(;
      L     MW 5158;
      T     MW 2078;
      SET;
      SAVE;
      CLR;
      A     BR;
      );
      JNB   _03a;
      L     MD 5160;
      DTR;
      T     #cv_re;
      SET;
      SAVE;
      CLR;
_03a: A     BR;
      );
      JNB   _03b;
      L     #cv_re;
      L     2.764800e+01;
      /R;
      T     #cv_re;
_03b: NOP   0;
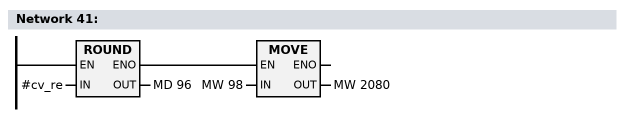
NETWORK
TITLE =
      A(;
      L     #cv_re;
      RND;
      T     MD 96;
      AN    OV;
      SAVE;
      CLR;
      A     BR;
      );
      JNB   _03c;
      L     MW 98;
      T     MW 2080;
_03c: NOP   0;
END_FUNCTION_BLOCK

// FB 58: know-how protected block, not included

// FC 105: know-how protected block, not included

// FC 106: know-how protected block, not included

DATA_BLOCK DB 1
VERSION : 0.0
"Pumps"
BEGIN
END_DATA_BLOCK

DATA_BLOCK DB 3
VERSION : 0.0
"Dat_CV_val"
BEGIN
END_DATA_BLOCK

DATA_BLOCK "COMM"	// DB 100
VERSION : 0.1
  STRUCT
   My_real_var : REAL ;
  END_STRUCT ;	
BEGIN
END_DATA_BLOCK

DATA_BLOCK "CV1_ctrl"	// DB 201
VERSION : 0.0
"klapan"
BEGIN
END_DATA_BLOCK

DATA_BLOCK "CV6_ctrl"	// DB 206
VERSION : 0.0
"klapan"
BEGIN
END_DATA_BLOCK

DATA_BLOCK "CV7_ctrl"	// DB 207
VERSION : 0.0
"klapan"
BEGIN
END_DATA_BLOCK

DATA_BLOCK "CV8_ctrl"	// DB 208
VERSION : 0.0
"klapan"
BEGIN
END_DATA_BLOCK

DATA_BLOCK "CV9_ctrl"	// DB 209
VERSION : 0.0
"klapan"
BEGIN
END_DATA_BLOCK

DATA_BLOCK "CV10_ctrl"	// DB 210
VERSION : 0.0
"klapan"
BEGIN
END_DATA_BLOCK

DATA_BLOCK "CV11_ctrl"	// DB 211
VERSION : 0.0
"klapan"
BEGIN
END_DATA_BLOCK

DATA_BLOCK "CV12_ctrl"	// DB 212
VERSION : 0.0
"klapan"
BEGIN
END_DATA_BLOCK

DATA_BLOCK "CV13_ctrl"	// DB 213
VERSION : 0.0
"klapan"
BEGIN
END_DATA_BLOCK

DATA_BLOCK "CV14_ctrl"	// DB 214
VERSION : 0.0
"klapan"
BEGIN
END_DATA_BLOCK

DATA_BLOCK "CV15_ctrl"	// DB 215
VERSION : 0.0
"klapan"
BEGIN
END_DATA_BLOCK

DATA_BLOCK "CV16_ctrl"	// DB 216
VERSION : 0.0
"klapan"
BEGIN
END_DATA_BLOCK

DATA_BLOCK "CV17_ctrl"	// DB 217
VERSION : 0.0
"klapan"
BEGIN
END_DATA_BLOCK

DATA_BLOCK "CV18_1_ctrl"	// DB 218
VERSION : 0.0
"klapan"
BEGIN
END_DATA_BLOCK

DATA_BLOCK "CV18_2_ctrl"	// DB 219
VERSION : 0.0
"klapan"
BEGIN
END_DATA_BLOCK

DATA_BLOCK "CV21_ctrl"	// DB 221
VERSION : 0.0
"klapan"
BEGIN
END_DATA_BLOCK

DATA_BLOCK "CV22_ctrl"	// DB 222
VERSION : 0.0
"klapan"
BEGIN
END_DATA_BLOCK

DATA_BLOCK "ctrl_CV23"	// DB 223
VERSION : 0.0
"klapan"
BEGIN
END_DATA_BLOCK

DATA_BLOCK "ctrl_CV24"	// DB 224
VERSION : 0.0
"klapan"
BEGIN
END_DATA_BLOCK

DATA_BLOCK "ctrl_CV25"	// DB 225
VERSION : 0.0
"klapan"
BEGIN
END_DATA_BLOCK

DATA_BLOCK "pid_cv1"	// DB 501
AUTHOR : SIMATIC
FAMILY : CONTROL
VERSION : 0.1
"TCONT_CP"
BEGIN
END_DATA_BLOCK

DATA_BLOCK "pid_cv2"	// DB 502
AUTHOR : SIMATIC
FAMILY : CONTROL
VERSION : 0.1
"TCONT_CP"
BEGIN
END_DATA_BLOCK

DATA_BLOCK DB 503
AUTHOR : SIMATIC
FAMILY : CONTROL
VERSION : 0.1
"TCONT_CP"
BEGIN
END_DATA_BLOCK

DATA_BLOCK "pid_cv6"	// DB 506
AUTHOR : SIMATIC
FAMILY : CONTROL
VERSION : 0.1
"TCONT_CP"
BEGIN
END_DATA_BLOCK

DATA_BLOCK "pid_cv7"	// DB 507
AUTHOR : SIMATIC
FAMILY : CONTROL
VERSION : 0.1
"TCONT_CP"
BEGIN
END_DATA_BLOCK

DATA_BLOCK "pid_cv8"	// DB 508
AUTHOR : SIMATIC
FAMILY : CONTROL
VERSION : 0.1
"TCONT_CP"
BEGIN
END_DATA_BLOCK

DATA_BLOCK "pid_cv9"	// DB 509
AUTHOR : SIMATIC
FAMILY : CONTROL
VERSION : 0.1
"TCONT_CP"
BEGIN
END_DATA_BLOCK

DATA_BLOCK "pid_cv10"	// DB 510
AUTHOR : SIMATIC
FAMILY : CONTROL
VERSION : 0.1
"TCONT_CP"
BEGIN
END_DATA_BLOCK

DATA_BLOCK "pid_cv11"	// DB 511
AUTHOR : SIMATIC
FAMILY : CONTROL
VERSION : 0.1
"TCONT_CP"
BEGIN
END_DATA_BLOCK

DATA_BLOCK "pid_cv12"	// DB 512
AUTHOR : SIMATIC
FAMILY : CONTROL
VERSION : 0.1
"TCONT_CP"
BEGIN
END_DATA_BLOCK

DATA_BLOCK "pid_cv13"	// DB 513
AUTHOR : SIMATIC
FAMILY : CONTROL
VERSION : 0.1
"TCONT_CP"
BEGIN
END_DATA_BLOCK

DATA_BLOCK "pid_cv14"	// DB 514
AUTHOR : SIMATIC
FAMILY : CONTROL
VERSION : 0.1
"TCONT_CP"
BEGIN
END_DATA_BLOCK

DATA_BLOCK "pid_cv15"	// DB 515
AUTHOR : SIMATIC
FAMILY : CONTROL
VERSION : 0.1
"TCONT_CP"
BEGIN
END_DATA_BLOCK

DATA_BLOCK "pid_cv16"	// DB 516
AUTHOR : SIMATIC
FAMILY : CONTROL
VERSION : 0.1
"TCONT_CP"
BEGIN
END_DATA_BLOCK

DATA_BLOCK "pid_cv17"	// DB 517
AUTHOR : SIMATIC
FAMILY : CONTROL
VERSION : 0.1
"TCONT_CP"
BEGIN
END_DATA_BLOCK

DATA_BLOCK "pid_cv18_1"	// DB 518
AUTHOR : SIMATIC
FAMILY : CONTROL
VERSION : 0.1
"TCONT_CP"
BEGIN
END_DATA_BLOCK

DATA_BLOCK "pid_cv18_2"	// DB 519
AUTHOR : SIMATIC
FAMILY : CONTROL
VERSION : 0.1
"TCONT_CP"
BEGIN
END_DATA_BLOCK

DATA_BLOCK "pid_cv21"	// DB 521
AUTHOR : SIMATIC
FAMILY : CONTROL
VERSION : 0.1
"TCONT_CP"
BEGIN
END_DATA_BLOCK

DATA_BLOCK "pid_cv22"	// DB 522
AUTHOR : SIMATIC
FAMILY : CONTROL
VERSION : 0.1
"TCONT_CP"
BEGIN
END_DATA_BLOCK

DATA_BLOCK "pid_cv23"	// DB 523
AUTHOR : SIMATIC
FAMILY : CONTROL
VERSION : 0.1
"TCONT_CP"
BEGIN
END_DATA_BLOCK

DATA_BLOCK "pid_cv24"	// DB 524
AUTHOR : SIMATIC
FAMILY : CONTROL
VERSION : 0.1
"TCONT_CP"
BEGIN
END_DATA_BLOCK

DATA_BLOCK "pid_cv25"	// DB 525
AUTHOR : SIMATIC
FAMILY : CONTROL
VERSION : 0.1
"TCONT_CP"
BEGIN
END_DATA_BLOCK

ORGANIZATION_BLOCK OB 1
TITLE = "Main Program Sweep (Cycle)"
VERSION : 0.1
VAR_TEMP
  OB1_EV_CLASS : BYTE ;	//Bits 0-3 = 1 (Coming event), Bits 4-7 = 1 (Event class 1)
  OB1_SCAN_1 : BYTE ;	//1 (Cold restart scan 1 of OB 1), 3 (Scan 2-n of OB 1)
  OB1_PRIORITY : BYTE ;	//Priority of OB Execution
  OB1_OB_NUMBR : BYTE ;	//1 (Organization block 1, OB1)
  OB1_RESERVED_1 : BYTE ;	//Reserved for system
  OB1_RESERVED_2 : BYTE ;	//Reserved for system
  OB1_PREV_CYCLE : INT ;	//Cycle time of previous OB1 scan (milliseconds)
  OB1_MIN_CYCLE : INT ;	//Minimum cycle time of OB1 (milliseconds)
  OB1_MAX_CYCLE : INT ;	//Maximum cycle time of OB1 (milliseconds)
  OB1_DATE_TIME : DATE_AND_TIME ;	//Date and time OB1 started
  bypass : BOOL ;
  bip : BOOL ;
  PT201 : REAL ;
  ret_avg10 : BOOL ;
  err_pt201 : BOOL ;
  err_pt203 : BOOL ;
  err_pt205 : BOOL ;
  err_pt206 : BOOL ;
  err_pt207 : BOOL ;
  err_pt208 : BOOL ;
  err_pt209 : BOOL ;
  err_pt210 : BOOL ;
  err_pt211 : BOOL ;
  err_pt212 : BOOL ;
  err_pt213 : BOOL ;
  err_pt214 : BOOL ;
  err_pt215 : BOOL ;
  err_lt301 : BOOL ;
  err_lt302 : BOOL ;
  err_lt303 : BOOL ;
  err_lt304 : BOOL ;
  LT301_re : REAL ;
  LT302_re : REAL ;
  LT303_re : REAL ;
  LT304_re : REAL ;
  err_pt202 : BOOL ;
  err_dpt216 : BOOL ;
  err_dpt217 : BOOL ;
  cv19_1_re : REAL ;
  fls : BOOL ;
  ret : WORD ;
  cv19_2_re : REAL ;
  doz_zasuv_re : REAL ;
END_VAR
BEGIN
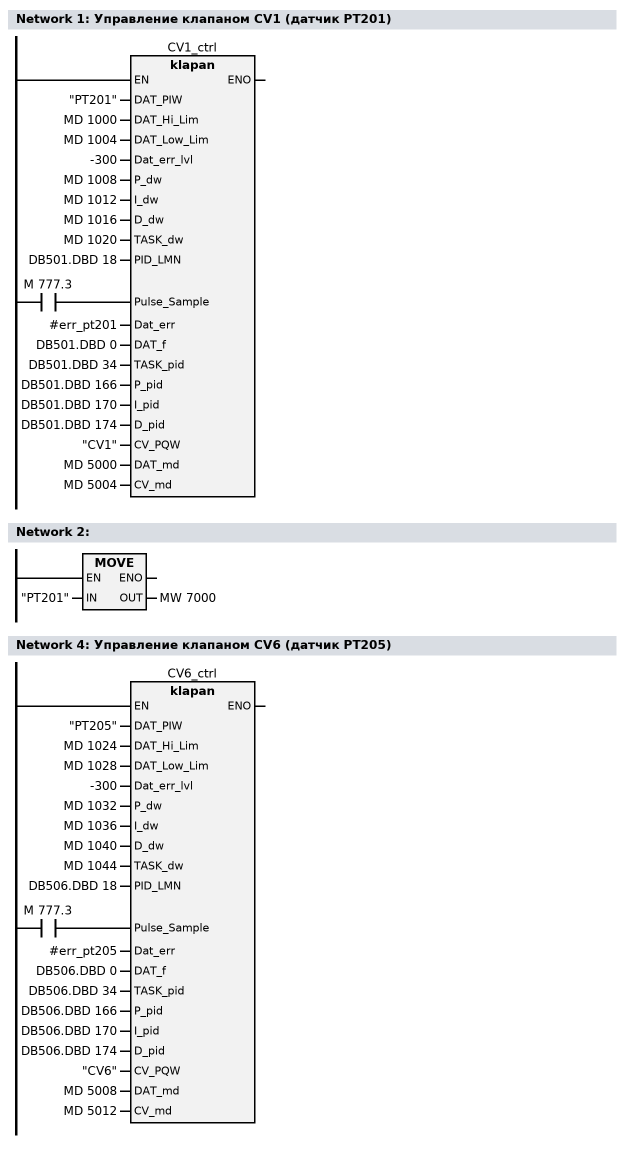
NETWORK
TITLE = Управление клапаном CV1 (датчик PT201)
      A     M 777.3;
      =     L 64.0;
      BLD   103;
      CALL  "klapan" , "CV1_ctrl" (
           DAT_PIW                  := "PT201",
           DAT_Hi_Lim               := MD 1000,
           DAT_Low_Lim              := MD 1004,
           Dat_err_lvl              := -300,
           P_dw                     := MD 1008,
           I_dw                     := MD 1012,
           D_dw                     := MD 1016,
           TASK_dw                  := MD 1020,
           PID_LMN                  := DB501.DBD 18,
           Pulse_Sample             := L 64.0,
           Dat_err                  := #err_pt201,
           DAT_f                    := DB501.DBD 0,
           TASK_pid                 := DB501.DBD 34,
           P_pid                    := DB501.DBD 166,
           I_pid                    := DB501.DBD 170,
           D_pid                    := DB501.DBD 174,
           CV_PQW                   := "CV1",
           DAT_md                   := MD 5000,
           CV_md                    := MD 5004);
      NOP   0;
NETWORK
TITLE =
      L     "PT201";
      T     MW 7000;
      NOP   0;
NETWORK
TITLE =
NETWORK
TITLE = Управление клапаном CV6 (датчик PT205)
      A     M 777.3;
      =     L 64.0;
      BLD   103;
      CALL  "klapan" , "CV6_ctrl" (
           DAT_PIW                  := "PT205",
           DAT_Hi_Lim               := MD 1024,
           DAT_Low_Lim              := MD 1028,
           Dat_err_lvl              := -300,
           P_dw                     := MD 1032,
           I_dw                     := MD 1036,
           D_dw                     := MD 1040,
           TASK_dw                  := MD 1044,
           PID_LMN                  := DB506.DBD 18,
           Pulse_Sample             := L 64.0,
           Dat_err                  := #err_pt205,
           DAT_f                    := DB506.DBD 0,
           TASK_pid                 := DB506.DBD 34,
           P_pid                    := DB506.DBD 166,
           I_pid                    := DB506.DBD 170,
           D_pid                    := DB506.DBD 174,
           CV_PQW                   := "CV6",
           DAT_md                   := MD 5008,
           CV_md                    := MD 5012);
      NOP   0;
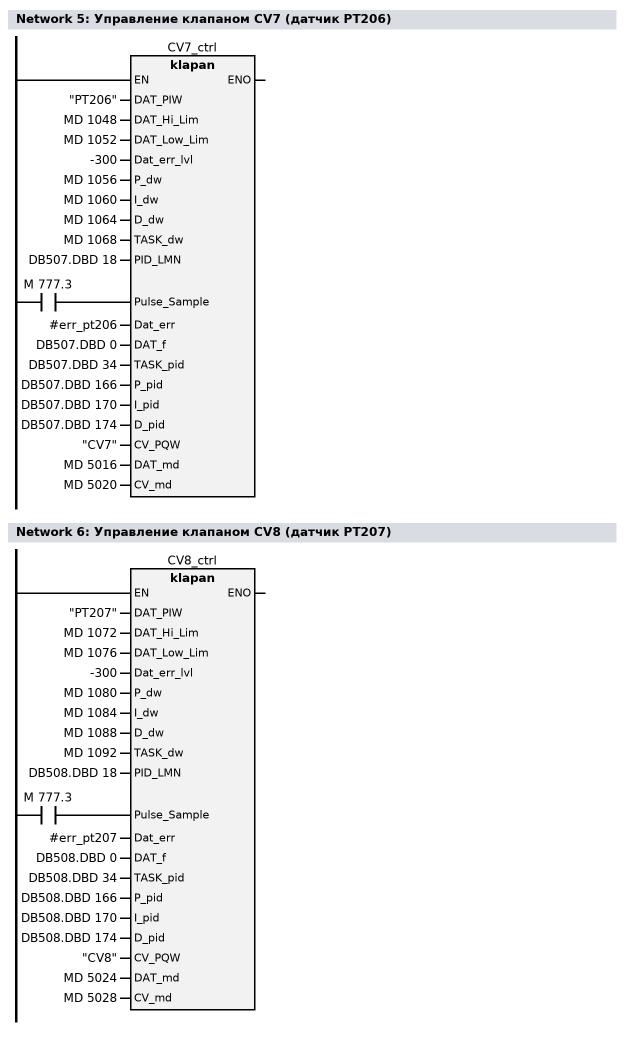
NETWORK
TITLE = Управление клапаном CV7 (датчик PT206)
      A     M 777.3;
      =     L 64.0;
      BLD   103;
      CALL  "klapan" , "CV7_ctrl" (
           DAT_PIW                  := "PT206",
           DAT_Hi_Lim               := MD 1048,
           DAT_Low_Lim              := MD 1052,
           Dat_err_lvl              := -300,
           P_dw                     := MD 1056,
           I_dw                     := MD 1060,
           D_dw                     := MD 1064,
           TASK_dw                  := MD 1068,
           PID_LMN                  := DB507.DBD 18,
           Pulse_Sample             := L 64.0,
           Dat_err                  := #err_pt206,
           DAT_f                    := DB507.DBD 0,
           TASK_pid                 := DB507.DBD 34,
           P_pid                    := DB507.DBD 166,
           I_pid                    := DB507.DBD 170,
           D_pid                    := DB507.DBD 174,
           CV_PQW                   := "CV7",
           DAT_md                   := MD 5016,
           CV_md                    := MD 5020);
      NOP   0;
NETWORK
TITLE = Управление клапаном CV8 (датчик PT207)
      A     M 777.3;
      =     L 64.0;
      BLD   103;
      CALL  "klapan" , "CV8_ctrl" (
           DAT_PIW                  := "PT207",
           DAT_Hi_Lim               := MD 1072,
           DAT_Low_Lim              := MD 1076,
           Dat_err_lvl              := -300,
           P_dw                     := MD 1080,
           I_dw                     := MD 1084,
           D_dw                     := MD 1088,
           TASK_dw                  := MD 1092,
           PID_LMN                  := DB508.DBD 18,
           Pulse_Sample             := L 64.0,
           Dat_err                  := #err_pt207,
           DAT_f                    := DB508.DBD 0,
           TASK_pid                 := DB508.DBD 34,
           P_pid                    := DB508.DBD 166,
           I_pid                    := DB508.DBD 170,
           D_pid                    := DB508.DBD 174,
           CV_PQW                   := "CV8",
           DAT_md                   := MD 5024,
           CV_md                    := MD 5028);
      NOP   0;
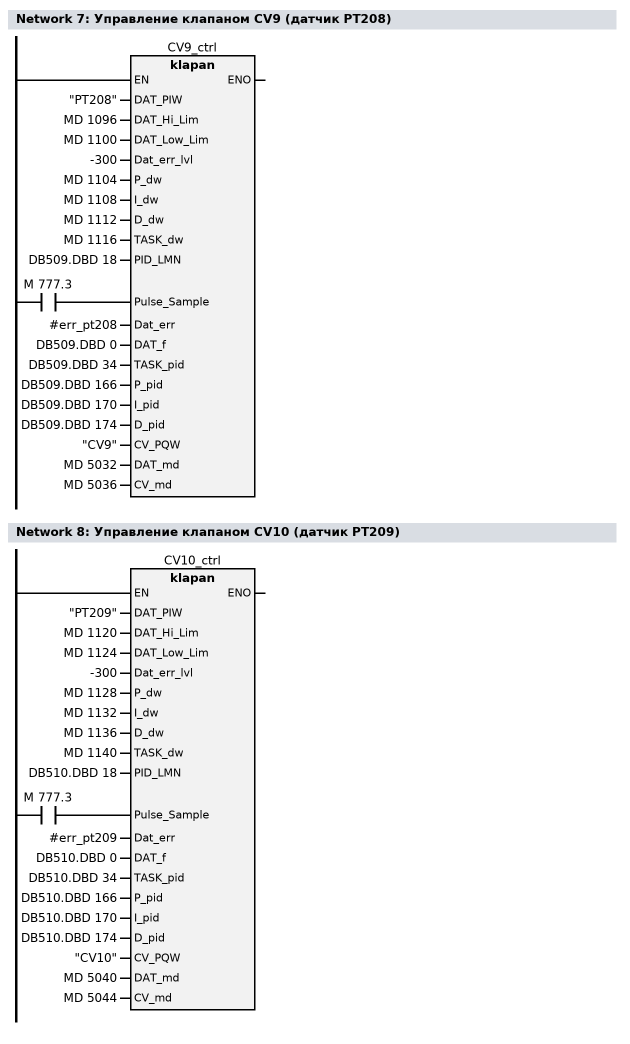
NETWORK
TITLE = Управление клапаном CV9 (датчик PT208)
      A     M 777.3;
      =     L 64.0;
      BLD   103;
      CALL  "klapan" , "CV9_ctrl" (
           DAT_PIW                  := "PT208",
           DAT_Hi_Lim               := MD 1096,
           DAT_Low_Lim              := MD 1100,
           Dat_err_lvl              := -300,
           P_dw                     := MD 1104,
           I_dw                     := MD 1108,
           D_dw                     := MD 1112,
           TASK_dw                  := MD 1116,
           PID_LMN                  := DB509.DBD 18,
           Pulse_Sample             := L 64.0,
           Dat_err                  := #err_pt208,
           DAT_f                    := DB509.DBD 0,
           TASK_pid                 := DB509.DBD 34,
           P_pid                    := DB509.DBD 166,
           I_pid                    := DB509.DBD 170,
           D_pid                    := DB509.DBD 174,
           CV_PQW                   := "CV9",
           DAT_md                   := MD 5032,
           CV_md                    := MD 5036);
      NOP   0;
NETWORK
TITLE = Управление клапаном CV10 (датчик PT209)
      A     M 777.3;
      =     L 64.0;
      BLD   103;
      CALL  "klapan" , "CV10_ctrl" (
           DAT_PIW                  := "PT209",
           DAT_Hi_Lim               := MD 1120,
           DAT_Low_Lim              := MD 1124,
           Dat_err_lvl              := -300,
           P_dw                     := MD 1128,
           I_dw                     := MD 1132,
           D_dw                     := MD 1136,
           TASK_dw                  := MD 1140,
           PID_LMN                  := DB510.DBD 18,
           Pulse_Sample             := L 64.0,
           Dat_err                  := #err_pt209,
           DAT_f                    := DB510.DBD 0,
           TASK_pid                 := DB510.DBD 34,
           P_pid                    := DB510.DBD 166,
           I_pid                    := DB510.DBD 170,
           D_pid                    := DB510.DBD 174,
           CV_PQW                   := "CV10",
           DAT_md                   := MD 5040,
           CV_md                    := MD 5044);
      NOP   0;
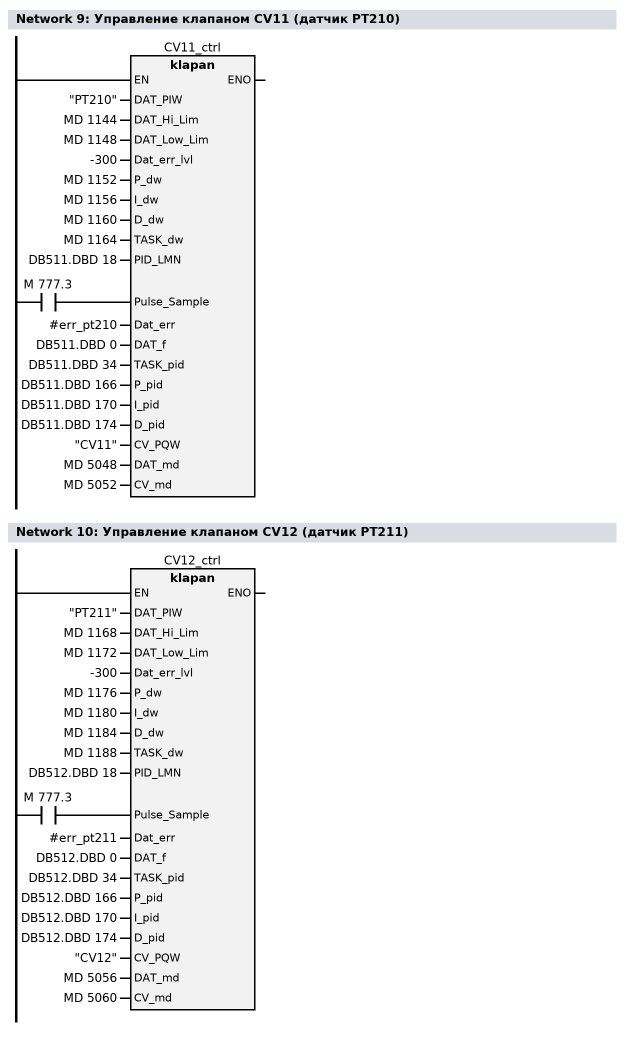
NETWORK
TITLE = Управление клапаном CV11 (датчик PT210)
      A     M 777.3;
      =     L 64.0;
      BLD   103;
      CALL  "klapan" , "CV11_ctrl" (
           DAT_PIW                  := "PT210",
           DAT_Hi_Lim               := MD 1144,
           DAT_Low_Lim              := MD 1148,
           Dat_err_lvl              := -300,
           P_dw                     := MD 1152,
           I_dw                     := MD 1156,
           D_dw                     := MD 1160,
           TASK_dw                  := MD 1164,
           PID_LMN                  := DB511.DBD 18,
           Pulse_Sample             := L 64.0,
           Dat_err                  := #err_pt210,
           DAT_f                    := DB511.DBD 0,
           TASK_pid                 := DB511.DBD 34,
           P_pid                    := DB511.DBD 166,
           I_pid                    := DB511.DBD 170,
           D_pid                    := DB511.DBD 174,
           CV_PQW                   := "CV11",
           DAT_md                   := MD 5048,
           CV_md                    := MD 5052);
      NOP   0;
NETWORK
TITLE = Управление клапаном CV12 (датчик PT211)
      A     M 777.3;
      =     L 64.0;
      BLD   103;
      CALL  "klapan" , "CV12_ctrl" (
           DAT_PIW                  := "PT211",
           DAT_Hi_Lim               := MD 1168,
           DAT_Low_Lim              := MD 1172,
           Dat_err_lvl              := -300,
           P_dw                     := MD 1176,
           I_dw                     := MD 1180,
           D_dw                     := MD 1184,
           TASK_dw                  := MD 1188,
           PID_LMN                  := DB512.DBD 18,
           Pulse_Sample             := L 64.0,
           Dat_err                  := #err_pt211,
           DAT_f                    := DB512.DBD 0,
           TASK_pid                 := DB512.DBD 34,
           P_pid                    := DB512.DBD 166,
           I_pid                    := DB512.DBD 170,
           D_pid                    := DB512.DBD 174,
           CV_PQW                   := "CV12",
           DAT_md                   := MD 5056,
           CV_md                    := MD 5060);
      NOP   0;
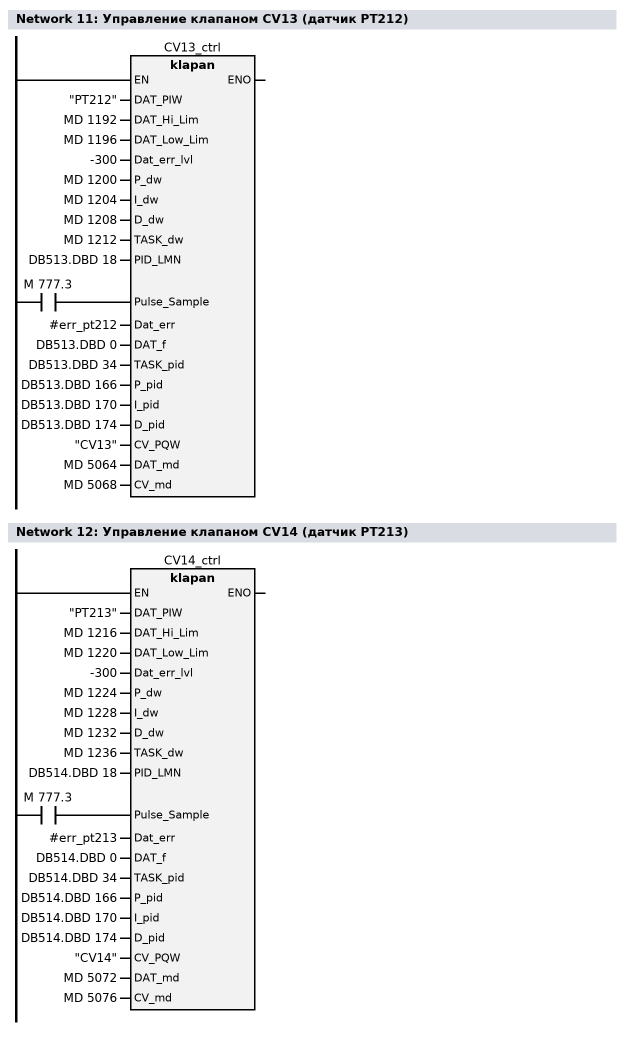
NETWORK
TITLE = Управление клапаном CV13 (датчик PT212)
      A     M 777.3;
      =     L 64.0;
      BLD   103;
      CALL  "klapan" , "CV13_ctrl" (
           DAT_PIW                  := "PT212",
           DAT_Hi_Lim               := MD 1192,
           DAT_Low_Lim              := MD 1196,
           Dat_err_lvl              := -300,
           P_dw                     := MD 1200,
           I_dw                     := MD 1204,
           D_dw                     := MD 1208,
           TASK_dw                  := MD 1212,
           PID_LMN                  := DB513.DBD 18,
           Pulse_Sample             := L 64.0,
           Dat_err                  := #err_pt212,
           DAT_f                    := DB513.DBD 0,
           TASK_pid                 := DB513.DBD 34,
           P_pid                    := DB513.DBD 166,
           I_pid                    := DB513.DBD 170,
           D_pid                    := DB513.DBD 174,
           CV_PQW                   := "CV13",
           DAT_md                   := MD 5064,
           CV_md                    := MD 5068);
      NOP   0;
NETWORK
TITLE = Управление клапаном CV14 (датчик PT213)
      A     M 777.3;
      =     L 64.0;
      BLD   103;
      CALL  "klapan" , "CV14_ctrl" (
           DAT_PIW                  := "PT213",
           DAT_Hi_Lim               := MD 1216,
           DAT_Low_Lim              := MD 1220,
           Dat_err_lvl              := -300,
           P_dw                     := MD 1224,
           I_dw                     := MD 1228,
           D_dw                     := MD 1232,
           TASK_dw                  := MD 1236,
           PID_LMN                  := DB514.DBD 18,
           Pulse_Sample             := L 64.0,
           Dat_err                  := #err_pt213,
           DAT_f                    := DB514.DBD 0,
           TASK_pid                 := DB514.DBD 34,
           P_pid                    := DB514.DBD 166,
           I_pid                    := DB514.DBD 170,
           D_pid                    := DB514.DBD 174,
           CV_PQW                   := "CV14",
           DAT_md                   := MD 5072,
           CV_md                    := MD 5076);
      NOP   0;
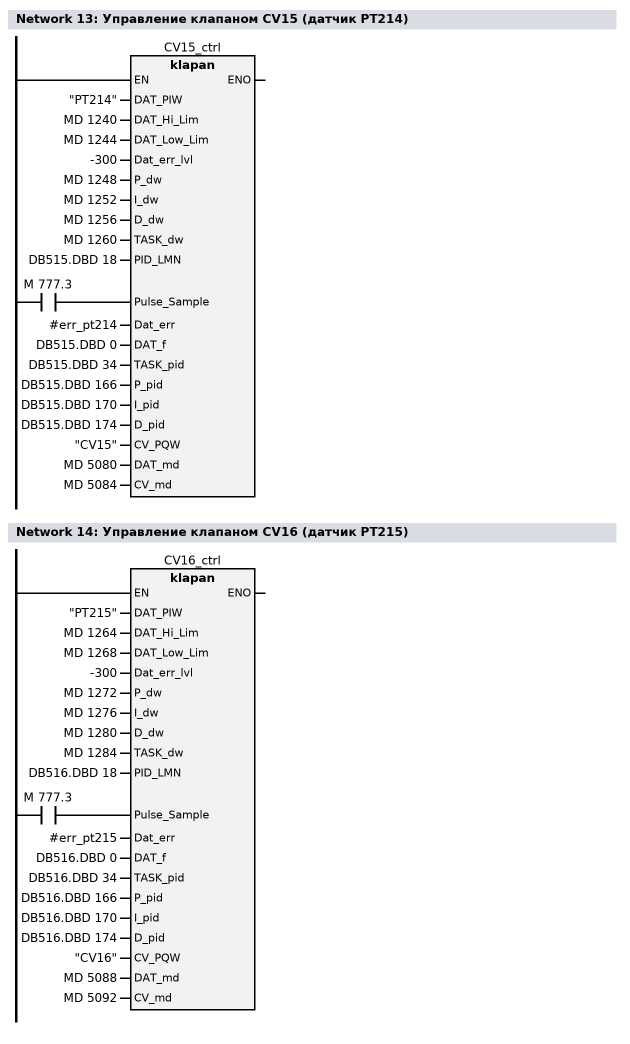
NETWORK
TITLE = Управление клапаном CV15 (датчик PT214)
      A     M 777.3;
      =     L 64.0;
      BLD   103;
      CALL  "klapan" , "CV15_ctrl" (
           DAT_PIW                  := "PT214",
           DAT_Hi_Lim               := MD 1240,
           DAT_Low_Lim              := MD 1244,
           Dat_err_lvl              := -300,
           P_dw                     := MD 1248,
           I_dw                     := MD 1252,
           D_dw                     := MD 1256,
           TASK_dw                  := MD 1260,
           PID_LMN                  := DB515.DBD 18,
           Pulse_Sample             := L 64.0,
           Dat_err                  := #err_pt214,
           DAT_f                    := DB515.DBD 0,
           TASK_pid                 := DB515.DBD 34,
           P_pid                    := DB515.DBD 166,
           I_pid                    := DB515.DBD 170,
           D_pid                    := DB515.DBD 174,
           CV_PQW                   := "CV15",
           DAT_md                   := MD 5080,
           CV_md                    := MD 5084);
      NOP   0;
NETWORK
TITLE = Управление клапаном CV16 (датчик PT215)
      A     M 777.3;
      =     L 64.0;
      BLD   103;
      CALL  "klapan" , "CV16_ctrl" (
           DAT_PIW                  := "PT215",
           DAT_Hi_Lim               := MD 1264,
           DAT_Low_Lim              := MD 1268,
           Dat_err_lvl              := -300,
           P_dw                     := MD 1272,
           I_dw                     := MD 1276,
           D_dw                     := MD 1280,
           TASK_dw                  := MD 1284,
           PID_LMN                  := DB516.DBD 18,
           Pulse_Sample             := L 64.0,
           Dat_err                  := #err_pt215,
           DAT_f                    := DB516.DBD 0,
           TASK_pid                 := DB516.DBD 34,
           P_pid                    := DB516.DBD 166,
           I_pid                    := DB516.DBD 170,
           D_pid                    := DB516.DBD 174,
           CV_PQW                   := "CV16",
           DAT_md                   := MD 5088,
           CV_md                    := MD 5092);
      NOP   0;
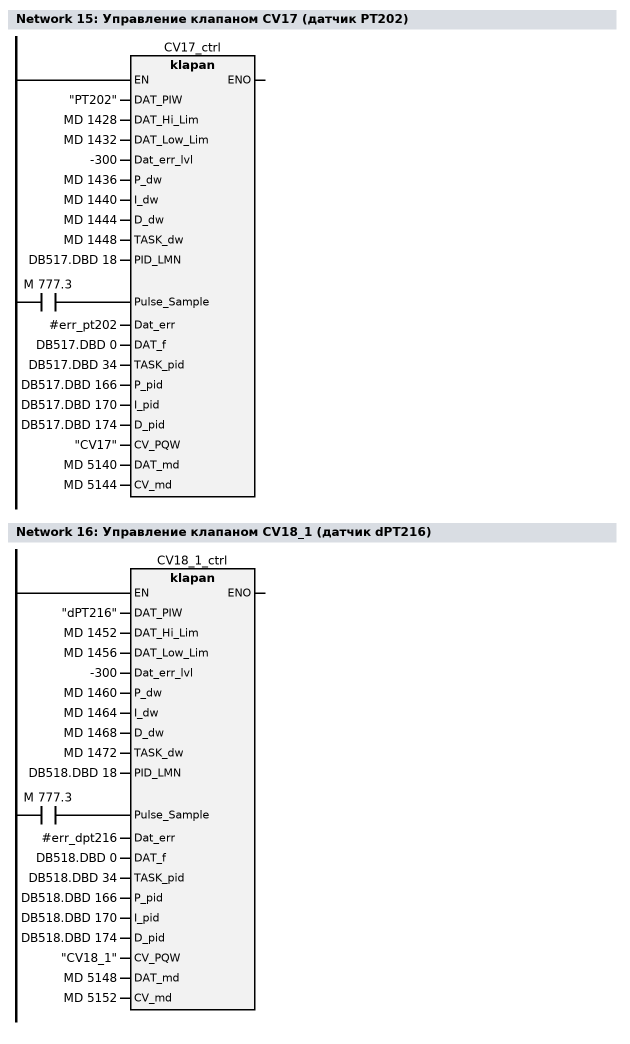
NETWORK
TITLE = Управление клапаном CV17 (датчик PT202)
      A     M 777.3;
      =     L 64.0;
      BLD   103;
      CALL  "klapan" , "CV17_ctrl" (
           DAT_PIW                  := "PT202",
           DAT_Hi_Lim               := MD 1428,
           DAT_Low_Lim              := MD 1432,
           Dat_err_lvl              := -300,
           P_dw                     := MD 1436,
           I_dw                     := MD 1440,
           D_dw                     := MD 1444,
           TASK_dw                  := MD 1448,
           PID_LMN                  := DB517.DBD 18,
           Pulse_Sample             := L 64.0,
           Dat_err                  := #err_pt202,
           DAT_f                    := DB517.DBD 0,
           TASK_pid                 := DB517.DBD 34,
           P_pid                    := DB517.DBD 166,
           I_pid                    := DB517.DBD 170,
           D_pid                    := DB517.DBD 174,
           CV_PQW                   := "CV17",
           DAT_md                   := MD 5140,
           CV_md                    := MD 5144);
      NOP   0;
NETWORK
TITLE = Управление клапаном CV18_1 (датчик dPT216)
      A     M 777.3;
      =     L 64.0;
      BLD   103;
      CALL  "klapan" , "CV18_1_ctrl" (
           DAT_PIW                  := "dPT216",
           DAT_Hi_Lim               := MD 1452,
           DAT_Low_Lim              := MD 1456,
           Dat_err_lvl              := -300,
           P_dw                     := MD 1460,
           I_dw                     := MD 1464,
           D_dw                     := MD 1468,
           TASK_dw                  := MD 1472,
           PID_LMN                  := DB518.DBD 18,
           Pulse_Sample             := L 64.0,
           Dat_err                  := #err_dpt216,
           DAT_f                    := DB518.DBD 0,
           TASK_pid                 := DB518.DBD 34,
           P_pid                    := DB518.DBD 166,
           I_pid                    := DB518.DBD 170,
           D_pid                    := DB518.DBD 174,
           CV_PQW                   := "CV18_1",
           DAT_md                   := MD 5148,
           CV_md                    := MD 5152);
      NOP   0;
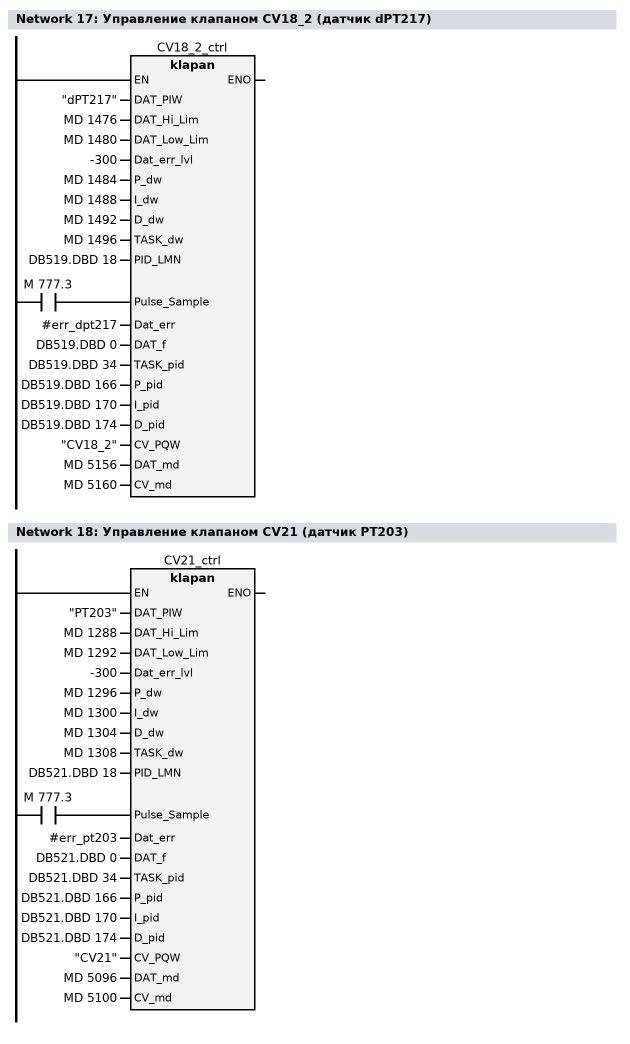
NETWORK
TITLE = Управление клапаном CV18_2 (датчик dPT217)
      A     M 777.3;
      =     L 64.0;
      BLD   103;
      CALL  "klapan" , "CV18_2_ctrl" (
           DAT_PIW                  := "dPT217",
           DAT_Hi_Lim               := MD 1476,
           DAT_Low_Lim              := MD 1480,
           Dat_err_lvl              := -300,
           P_dw                     := MD 1484,
           I_dw                     := MD 1488,
           D_dw                     := MD 1492,
           TASK_dw                  := MD 1496,
           PID_LMN                  := DB519.DBD 18,
           Pulse_Sample             := L 64.0,
           Dat_err                  := #err_dpt217,
           DAT_f                    := DB519.DBD 0,
           TASK_pid                 := DB519.DBD 34,
           P_pid                    := DB519.DBD 166,
           I_pid                    := DB519.DBD 170,
           D_pid                    := DB519.DBD 174,
           CV_PQW                   := "CV18_2",
           DAT_md                   := MD 5156,
           CV_md                    := MD 5160);
      NOP   0;
NETWORK
TITLE = Управление клапаном CV21 (датчик PT203)
      A     M 777.3;
      =     L 64.0;
      BLD   103;
      CALL  "klapan" , "CV21_ctrl" (
           DAT_PIW                  := "PT203",
           DAT_Hi_Lim               := MD 1288,
           DAT_Low_Lim              := MD 1292,
           Dat_err_lvl              := -300,
           P_dw                     := MD 1296,
           I_dw                     := MD 1300,
           D_dw                     := MD 1304,
           TASK_dw                  := MD 1308,
           PID_LMN                  := DB521.DBD 18,
           Pulse_Sample             := L 64.0,
           Dat_err                  := #err_pt203,
           DAT_f                    := DB521.DBD 0,
           TASK_pid                 := DB521.DBD 34,
           P_pid                    := DB521.DBD 166,
           I_pid                    := DB521.DBD 170,
           D_pid                    := DB521.DBD 174,
           CV_PQW                   := "CV21",
           DAT_md                   := MD 5096,
           CV_md                    := MD 5100);
      NOP   0;
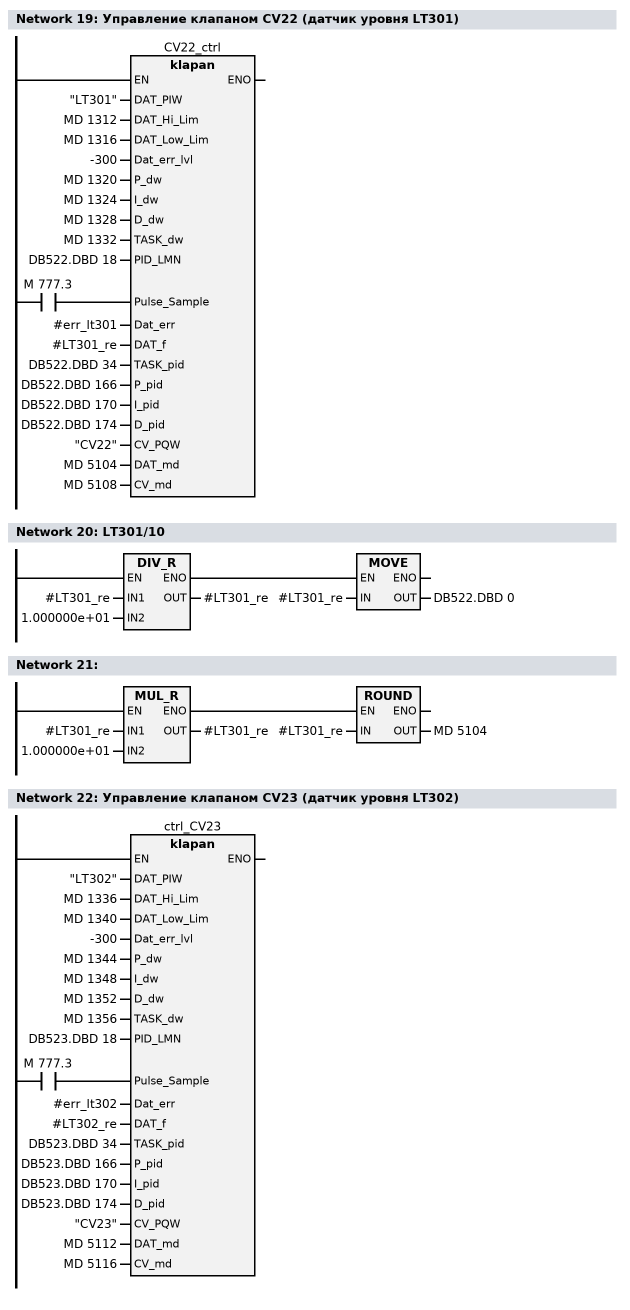
NETWORK
TITLE = Управление клапаном CV22 (датчик уровня LT301)
      A     M 777.3;
      =     L 64.0;
      BLD   103;
      CALL  "klapan" , "CV22_ctrl" (
           DAT_PIW                  := "LT301",
           DAT_Hi_Lim               := MD 1312,
           DAT_Low_Lim              := MD 1316,
           Dat_err_lvl              := -300,
           P_dw                     := MD 1320,
           I_dw                     := MD 1324,
           D_dw                     := MD 1328,
           TASK_dw                  := MD 1332,
           PID_LMN                  := DB522.DBD 18,
           Pulse_Sample             := L 64.0,
           Dat_err                  := #err_lt301,
           DAT_f                    := #LT301_re,
           TASK_pid                 := DB522.DBD 34,
           P_pid                    := DB522.DBD 166,
           I_pid                    := DB522.DBD 170,
           D_pid                    := DB522.DBD 174,
           CV_PQW                   := "CV22",
           DAT_md                   := MD 5104,
           CV_md                    := MD 5108);
      NOP   0;
NETWORK
TITLE = LT301/10
      A(;
      L     #LT301_re;
      L     1.000000e+01;
      /R;
      T     #LT301_re;
      AN    OV;
      SAVE;
      CLR;
      A     BR;
      );
      JNB   _001;
      L     #LT301_re;
      T     DB522.DBD 0;
_001: NOP   0;
NETWORK
TITLE =
      A(;
      L     #LT301_re;
      L     1.000000e+01;
      *R;
      T     #LT301_re;
      AN    OV;
      SAVE;
      CLR;
      A     BR;
      );
      JNB   _002;
      L     #LT301_re;
      RND;
      T     MD 5104;
_002: NOP   0;
NETWORK
TITLE = Управление клапаном CV23 (датчик уровня LT302)
      A     M 777.3;
      =     L 64.0;
      BLD   103;
      CALL  "klapan" , "ctrl_CV23" (
           DAT_PIW                  := "LT302",
           DAT_Hi_Lim               := MD 1336,
           DAT_Low_Lim              := MD 1340,
           Dat_err_lvl              := -300,
           P_dw                     := MD 1344,
           I_dw                     := MD 1348,
           D_dw                     := MD 1352,
           TASK_dw                  := MD 1356,
           PID_LMN                  := DB523.DBD 18,
           Pulse_Sample             := L 64.0,
           Dat_err                  := #err_lt302,
           DAT_f                    := #LT302_re,
           TASK_pid                 := DB523.DBD 34,
           P_pid                    := DB523.DBD 166,
           I_pid                    := DB523.DBD 170,
           D_pid                    := DB523.DBD 174,
           CV_PQW                   := "CV23",
           DAT_md                   := MD 5112,
           CV_md                    := MD 5116);
      NOP   0;
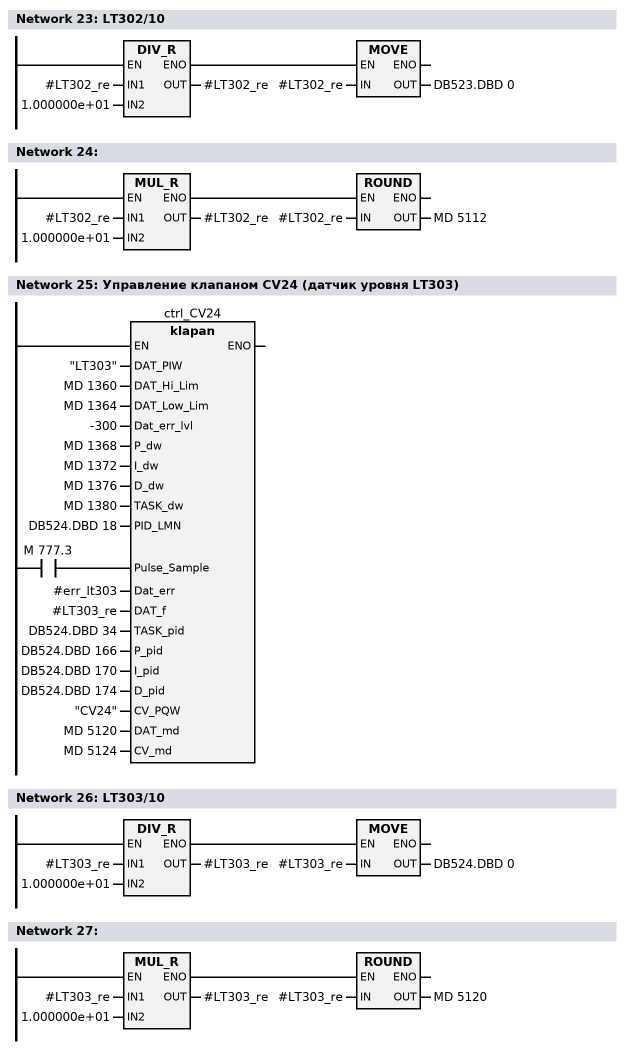
NETWORK
TITLE = LT302/10
      A(;
      L     #LT302_re;
      L     1.000000e+01;
      /R;
      T     #LT302_re;
      AN    OV;
      SAVE;
      CLR;
      A     BR;
      );
      JNB   _003;
      L     #LT302_re;
      T     DB523.DBD 0;
_003: NOP   0;
NETWORK
TITLE =
      A(;
      L     #LT302_re;
      L     1.000000e+01;
      *R;
      T     #LT302_re;
      AN    OV;
      SAVE;
      CLR;
      A     BR;
      );
      JNB   _004;
      L     #LT302_re;
      RND;
      T     MD 5112;
_004: NOP   0;
NETWORK
TITLE = Управление клапаном CV24 (датчик уровня LT303)
      A     M 777.3;
      =     L 64.0;
      BLD   103;
      CALL  "klapan" , "ctrl_CV24" (
           DAT_PIW                  := "LT303",
           DAT_Hi_Lim               := MD 1360,
           DAT_Low_Lim              := MD 1364,
           Dat_err_lvl              := -300,
           P_dw                     := MD 1368,
           I_dw                     := MD 1372,
           D_dw                     := MD 1376,
           TASK_dw                  := MD 1380,
           PID_LMN                  := DB524.DBD 18,
           Pulse_Sample             := L 64.0,
           Dat_err                  := #err_lt303,
           DAT_f                    := #LT303_re,
           TASK_pid                 := DB524.DBD 34,
           P_pid                    := DB524.DBD 166,
           I_pid                    := DB524.DBD 170,
           D_pid                    := DB524.DBD 174,
           CV_PQW                   := "CV24",
           DAT_md                   := MD 5120,
           CV_md                    := MD 5124);
      NOP   0;
NETWORK
TITLE = LT303/10
      A(;
      L     #LT303_re;
      L     1.000000e+01;
      /R;
      T     #LT303_re;
      AN    OV;
      SAVE;
      CLR;
      A     BR;
      );
      JNB   _005;
      L     #LT303_re;
      T     DB524.DBD 0;
_005: NOP   0;
NETWORK
TITLE =
      A(;
      L     #LT303_re;
      L     1.000000e+01;
      *R;
      T     #LT303_re;
      AN    OV;
      SAVE;
      CLR;
      A     BR;
      );
      JNB   _006;
      L     #LT303_re;
      RND;
      T     MD 5120;
_006: NOP   0;
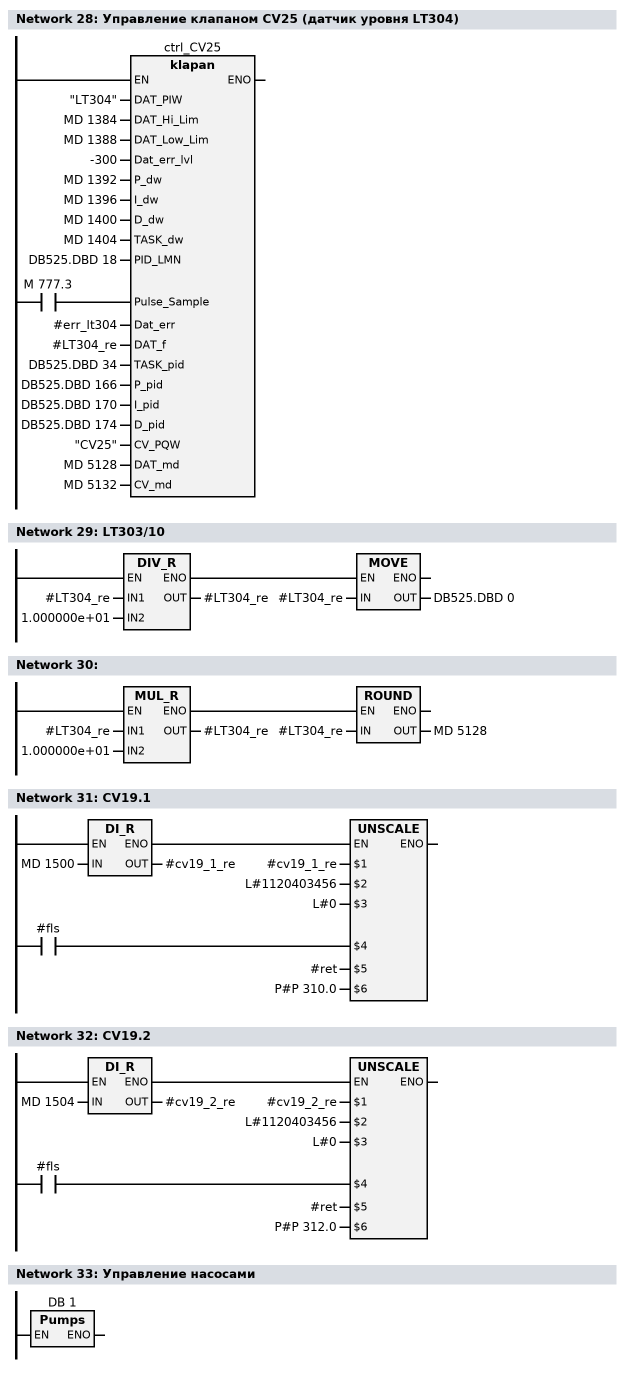
NETWORK
TITLE = Управление клапаном CV25 (датчик уровня LT304)
      A     M 777.3;
      =     L 64.0;
      BLD   103;
      CALL  "klapan" , "ctrl_CV25" (
           DAT_PIW                  := "LT304",
           DAT_Hi_Lim               := MD 1384,
           DAT_Low_Lim              := MD 1388,
           Dat_err_lvl              := -300,
           P_dw                     := MD 1392,
           I_dw                     := MD 1396,
           D_dw                     := MD 1400,
           TASK_dw                  := MD 1404,
           PID_LMN                  := DB525.DBD 18,
           Pulse_Sample             := L 64.0,
           Dat_err                  := #err_lt304,
           DAT_f                    := #LT304_re,
           TASK_pid                 := DB525.DBD 34,
           P_pid                    := DB525.DBD 166,
           I_pid                    := DB525.DBD 170,
           D_pid                    := DB525.DBD 174,
           CV_PQW                   := "CV25",
           DAT_md                   := MD 5128,
           CV_md                    := MD 5132);
      NOP   0;
NETWORK
TITLE = LT303/10
      A(;
      L     #LT304_re;
      L     1.000000e+01;
      /R;
      T     #LT304_re;
      AN    OV;
      SAVE;
      CLR;
      A     BR;
      );
      JNB   _007;
      L     #LT304_re;
      T     DB525.DBD 0;
_007: NOP   0;
NETWORK
TITLE =
      A(;
      L     #LT304_re;
      L     1.000000e+01;
      *R;
      T     #LT304_re;
      AN    OV;
      SAVE;
      CLR;
      A     BR;
      );
      JNB   _008;
      L     #LT304_re;
      RND;
      T     MD 5128;
_008: NOP   0;
NETWORK
TITLE = CV19.1
      A     #fls;
      =     L 64.0;
      BLD   103;
      A(;
      L     MD 1500;
      DTR;
      T     #cv19_1_re;
      SET;
      SAVE;
      CLR;
      A     BR;
      );
      JNB   _009;
      CALL  "UNSCALE" (
           $1                       := #cv19_1_re,
           $2                       := L#1120403456,
           $3                       := L#0,
           $4                       := L 64.0,
           $5                       := #ret,
           $6                       := P#P 310.0);
_009: NOP   0;
NETWORK
TITLE = CV19.2
      A     #fls;
      =     L 64.0;
      BLD   103;
      A(;
      L     MD 1504;
      DTR;
      T     #cv19_2_re;
      SET;
      SAVE;
      CLR;
      A     BR;
      );
      JNB   _00a;
      CALL  "UNSCALE" (
           $1                       := #cv19_2_re,
           $2                       := L#1120403456,
           $3                       := L#0,
           $4                       := L 64.0,
           $5                       := #ret,
           $6                       := P#P 312.0);
_00a: NOP   0;
NETWORK
TITLE = Управление насосами
      CALL  "Pumps" , DB 1;
      NOP   0;
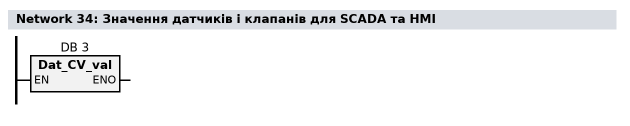
NETWORK
TITLE = Значення датчиків і клапанів для SCADA та HMI
      CALL  "Dat_CV_val" , DB 3;
      NOP   0;
END_ORGANIZATION_BLOCK

ORGANIZATION_BLOCK "CYC_INT5"	// OB 35
TITLE = "Cyclic Interrupt"
VERSION : 0.1
VAR_TEMP
  OB35_EV_CLASS : BYTE ;	//Bits 0-3 = 1 (Coming event), Bits 4-7 = 1 (Event class 1)
  OB35_STRT_INF : BYTE ;	//16#36 (OB 35 has started)
  OB35_PRIORITY : BYTE ;	//Priority of OB Execution
  OB35_OB_NUMBR : BYTE ;	//35 (Organization block 35, OB35)
  OB35_RESERVED_1 : BYTE ;	//Reserved for system
  OB35_RESERVED_2 : BYTE ;	//Reserved for system
  OB35_PHASE_OFFSET : WORD ;	//Phase offset (msec)
  OB35_RESERVED_3 : INT ;	//Reserved for system
  OB35_EXC_FREQ : INT ;	//Frequency of execution (msec)
  OB35_DATE_TIME : DATE_AND_TIME ;	//Date and time OB35 started
END_VAR
BEGIN
